//to Garlic
      O     "Blend_T-41".Dose_Garlic.QDOSERun;  //Dose Run
      =     "Blend to Preparation"."T-41".Raw_Material.Garlic.DoseRun;
      O     "Blend_T-41".Dose_Garlic.QHELD;  //Dose Held
      =     "Blend to Preparation"."T-41".Raw_Material.Garlic.DoseHeld;
      O     "Blend_T-41".Dose_Garlic.QDoseComplete;  //Dose Complete
      =     "Blend to Preparation"."T-41".Raw_Material.Garlic.DoseComplete;
      O     "Blend_T-41".Dose_Garlic.V_CMD;  //Valve Command
      =     "Blend to Preparation"."T-41".Raw_Material.Garlic.ValveCMD;
      O     "Blend_T-41".Dose_Garlic.P_CMD;  //Pump Command
      =     "Blend to Preparation"."T-41".Raw_Material.Garlic.PumpCMD;
      O     "Blend_T-41".Dose.Dose_Header_Req.%X7;  //Header 1 Req
      =     "Blend to Preparation"."T-41".Raw_Material.Garlic.Header1_Req;
      O     "Blend_T-41".Dose.Dose_Header_Req.%X23;  //Header 2 Req
      =     "Blend to Preparation"."T-41".Raw_Material.Garlic.Header2_Req;
      L     "Blend to Preparation".Recipe."T-41".Garlic.Sp_DoseQty;  //Load Sp Dose From Recipe
      T     "Blend_T-41".SP_Garlic.Dose_SP;
      L     "Blend_T-41".Dose_Garlic.P_SPEED;  //Pump Speed
      T     "Blend to Preparation".Recipe."T-41".Garlic.SP_PumpSpeed;

//to Vinegar
      O     "Blend_T-41".Dose_Vinegar.QDOSERun;  //Dose Run
      =     "Blend to Preparation"."T-41".Raw_Material.Vinegar.DoseRun;
      O     "Blend_T-41".Dose_Vinegar.QHELD;  //Dose Held
      =     "Blend to Preparation"."T-41".Raw_Material.Vinegar.DoseHeld;
      O     "Blend_T-41".Dose_Vinegar.QDoseComplete;  //Dose Complete
      =     "Blend to Preparation"."T-41".Raw_Material.Vinegar.DoseComplete;
      O     "Blend_T-41".Dose_Vinegar.V_CMD;  //Valve Command
      =     "Blend to Preparation"."T-41".Raw_Material.Vinegar.ValveCMD;
      O     "Blend_T-41".Dose_Vinegar.P_CMD;  //Pump Command
      =     "Blend to Preparation"."T-41".Raw_Material.Vinegar.PumpCMD;
      L     "Blend to Preparation".Recipe."T-41".Vinegar.Sp_DoseQty;  //Load Sp Dose From Recipe
      T     "Blend_T-41".SP_Vinegar.Dose_SP;
      L     "Blend_T-41".Dose_Vinegar.P_SPEED;  //Pump Speed
      T     "Blend to Preparation".Recipe."T-41".Vinegar.SP_PumpSpeed;

//to HW
      O     "Blend_T-41".Dose_HW.QDOSERun;  //Dose Run
      =     "Blend to Preparation"."T-41".Raw_Material.HW.DoseRun;
      O     "Blend_T-41".Dose_HW.QHELD;  //Dose Held
      =     "Blend to Preparation"."T-41".Raw_Material.HW.DoseHeld;
      O     "Blend_T-41".Dose_HW.QDoseComplete;  //Dose Complete
      =     "Blend to Preparation"."T-41".Raw_Material.HW.DoseComplete;
      O     "Blend_T-41".Dose_HW.V_CMD;  //Valve Command
      =     "Blend to Preparation"."T-41".Raw_Material.HW.ValveCMD;
      O     "Blend_T-41".Dose_HW.P_CMD;  //Pump Command
      =     "Blend to Preparation"."T-41".Raw_Material.HW.PumpCMD;
      O     "Blend_T-41".Dose.Dose_Header_Req.%X8;  //Header 1 Req
      =     "Blend to Preparation"."T-41".Raw_Material.HW.Header1_Req;
      O     "Blend_T-41".Dose.Dose_Header_Req.%X24;  //Header 2 Req
      =     "Blend to Preparation"."T-41".Raw_Material.HW.Header2_Req;

      L     "Blend to Preparation".Recipe."T-41".HW.Sp_Flush_to_BlendQty;  //Load Flush to Blend Sp Dose From Recipe
      T     "Blend_T-41"."HW Flushing".Qty."Flush to Blend Qty";
      L     "Blend to Preparation".Recipe."T-41".HW.Sp_Flush_to_DrainQty;  //Load Flush to Blend Sp Dose From Recipe
      T     "Blend_T-41"."HW Flushing".Qty."Flush to Drain Qty";  //Load Drain Time from recipe
      L     "Blend to Preparation".Recipe."T-41".HW.Sp_DrainTime;
      T     "Blend_T-41"."HW Flushing".TimeDrain_SP;

      L     "Blend_T-41".Dose_HW.P_SPEED;  //Pump Speed
      T     "Blend to Preparation".Recipe."T-41".HW.SP_PumpSpeed;


//General
      O     "Blend_T-41".IN_FBAV_Header1;
      =     "Blend to Preparation"."T-41".LineHeader1_OK;
      O     "Blend_T-41".IN_FBAV_Header2;
      =     "Blend to Preparation"."T-41".LineHeader2_OK;
      O     "Blend_T-41".IN_FBAV_Vinegar;
      =     "Blend to Preparation"."T-41".LineVinegar_OK;


REGION Network 124: Comm to Salt
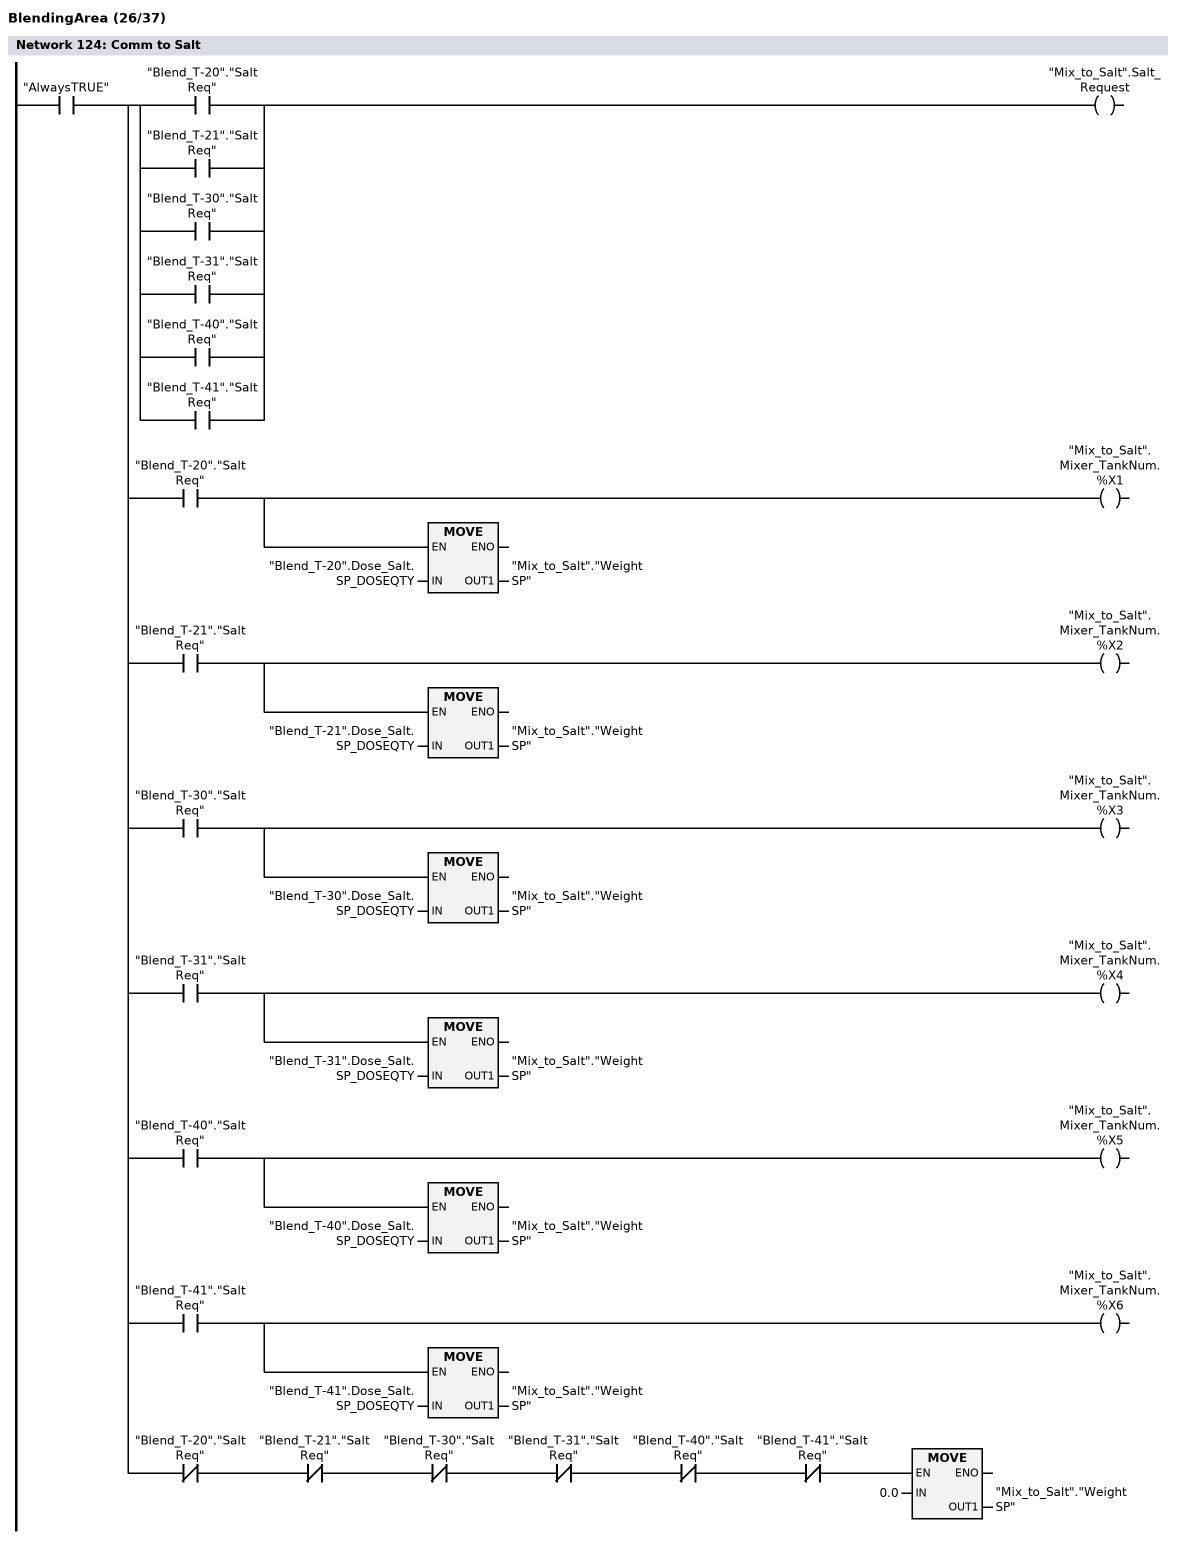
   RUNG wire#powerrail
      Contact( "AlwaysTRUE" )
      wire#w1
      Contact( "Blend_T-20"."Salt Req" )
      wire#w2
      Coil( "Mix_to_Salt".Salt_Request )
   END_RUNG
   RUNG wire#w1
      Contact( "Blend_T-21"."Salt Req" )
   END_RUNG wire#w2
   RUNG wire#w1
      Contact( "Blend_T-30"."Salt Req" )
   END_RUNG wire#w2
   RUNG wire#w1
      Contact( "Blend_T-31"."Salt Req" )
   END_RUNG wire#w2
   RUNG wire#w1
      Contact( "Blend_T-40"."Salt Req" )
   END_RUNG wire#w2
   RUNG wire#w1
      Contact( "Blend_T-41"."Salt Req" )
   END_RUNG wire#w2
   RUNG wire#w1
      Contact( "Blend_T-20"."Salt Req" )
      wire#w3
      Coil( "Mix_to_Salt".Mixer_TankNum.%X1 )
   END_RUNG
   RUNG wire#w3
      Move(in := "Blend_T-20".Dose_Salt.SP_DOSEQTY, out1 => "Mix_to_Salt"."Weight SP")
   END_RUNG
   RUNG wire#w1
      Contact( "Blend_T-21"."Salt Req" )
      wire#w4
      Coil( "Mix_to_Salt".Mixer_TankNum.%X2 )
   END_RUNG
   RUNG wire#w4
      Move(in := "Blend_T-21".Dose_Salt.SP_DOSEQTY, out1 => "Mix_to_Salt"."Weight SP")
   END_RUNG
   RUNG wire#w1
      Contact( "Blend_T-30"."Salt Req" )
      wire#w5
      Coil( "Mix_to_Salt".Mixer_TankNum.%X3 )
   END_RUNG
   RUNG wire#w5
      Move(in := "Blend_T-30".Dose_Salt.SP_DOSEQTY, out1 => "Mix_to_Salt"."Weight SP")
   END_RUNG
   RUNG wire#w1
      Contact( "Blend_T-31"."Salt Req" )
      wire#w6
      Coil( "Mix_to_Salt".Mixer_TankNum.%X4 )
   END_RUNG
   RUNG wire#w6
      Move(in := "Blend_T-31".Dose_Salt.SP_DOSEQTY, out1 => "Mix_to_Salt"."Weight SP")
   END_RUNG
   RUNG wire#w1
      Contact( "Blend_T-40"."Salt Req" )
      wire#w7
      Coil( "Mix_to_Salt".Mixer_TankNum.%X5 )
   END_RUNG
   RUNG wire#w7
      Move(in := "Blend_T-40".Dose_Salt.SP_DOSEQTY, out1 => "Mix_to_Salt"."Weight SP")
   END_RUNG
   RUNG wire#w1
      Contact( "Blend_T-41"."Salt Req" )
      wire#w8
      Coil( "Mix_to_Salt".Mixer_TankNum.%X6 )
   END_RUNG
   RUNG wire#w8
      Move(in := "Blend_T-41".Dose_Salt.SP_DOSEQTY, out1 => "Mix_to_Salt"."Weight SP")
   END_RUNG
   RUNG wire#w1
      I_Contact( "Blend_T-20"."Salt Req" )
      I_Contact( "Blend_T-21"."Salt Req" )
      I_Contact( "Blend_T-30"."Salt Req" )
      I_Contact( "Blend_T-31"."Salt Req" )
      I_Contact( "Blend_T-40"."Salt Req" )
      I_Contact( "Blend_T-41"."Salt Req" )
      Move(in := 0.0, out1 => "Mix_to_Salt"."Weight SP")
   END_RUNG
   // the same network as SCL:
   "Mix_to_Salt".Salt_Request := "AlwaysTRUE" AND ("Blend_T-20"."Salt Req" OR "Blend_T-21"."Salt Req" OR "Blend_T-30"."Salt Req" OR "Blend_T-31"."Salt Req" OR "Blend_T-40"."Salt Req" OR "Blend_T-41"."Salt Req");
   "Mix_to_Salt".Mixer_TankNum.%X1 := "AlwaysTRUE" AND "Blend_T-20"."Salt Req";
   IF "Mix_to_Salt".Mixer_TankNum.%X1 THEN
       "Mix_to_Salt"."Weight SP" := "Blend_T-20".Dose_Salt.SP_DOSEQTY;
   END_IF;
   "Mix_to_Salt".Mixer_TankNum.%X2 := "AlwaysTRUE" AND "Blend_T-21"."Salt Req";
   IF "Mix_to_Salt".Mixer_TankNum.%X2 THEN
       "Mix_to_Salt"."Weight SP" := "Blend_T-21".Dose_Salt.SP_DOSEQTY;
   END_IF;
   "Mix_to_Salt".Mixer_TankNum.%X3 := "AlwaysTRUE" AND "Blend_T-30"."Salt Req";
   IF "Mix_to_Salt".Mixer_TankNum.%X3 THEN
       "Mix_to_Salt"."Weight SP" := "Blend_T-30".Dose_Salt.SP_DOSEQTY;
   END_IF;
   "Mix_to_Salt".Mixer_TankNum.%X4 := "AlwaysTRUE" AND "Blend_T-31"."Salt Req";
   IF "Mix_to_Salt".Mixer_TankNum.%X4 THEN
       "Mix_to_Salt"."Weight SP" := "Blend_T-31".Dose_Salt.SP_DOSEQTY;
   END_IF;
   "Mix_to_Salt".Mixer_TankNum.%X5 := "AlwaysTRUE" AND "Blend_T-40"."Salt Req";
   IF "Mix_to_Salt".Mixer_TankNum.%X5 THEN
       "Mix_to_Salt"."Weight SP" := "Blend_T-40".Dose_Salt.SP_DOSEQTY;
   END_IF;
   "Mix_to_Salt".Mixer_TankNum.%X6 := "AlwaysTRUE" AND "Blend_T-41"."Salt Req";
   IF "Mix_to_Salt".Mixer_TankNum.%X6 THEN
       "Mix_to_Salt"."Weight SP" := "Blend_T-41".Dose_Salt.SP_DOSEQTY;
   END_IF;
   IF "AlwaysTRUE" AND NOT "Blend_T-20"."Salt Req" AND NOT "Blend_T-21"."Salt Req" AND NOT "Blend_T-30"."Salt Req" AND NOT "Blend_T-31"."Salt Req" AND NOT "Blend_T-40"."Salt Req" AND NOT "Blend_T-41"."Salt Req" THEN
       "Mix_to_Salt"."Weight SP" := 0.0;
   END_IF;
END_REGION

REGION Network 125: Comm to Sugar
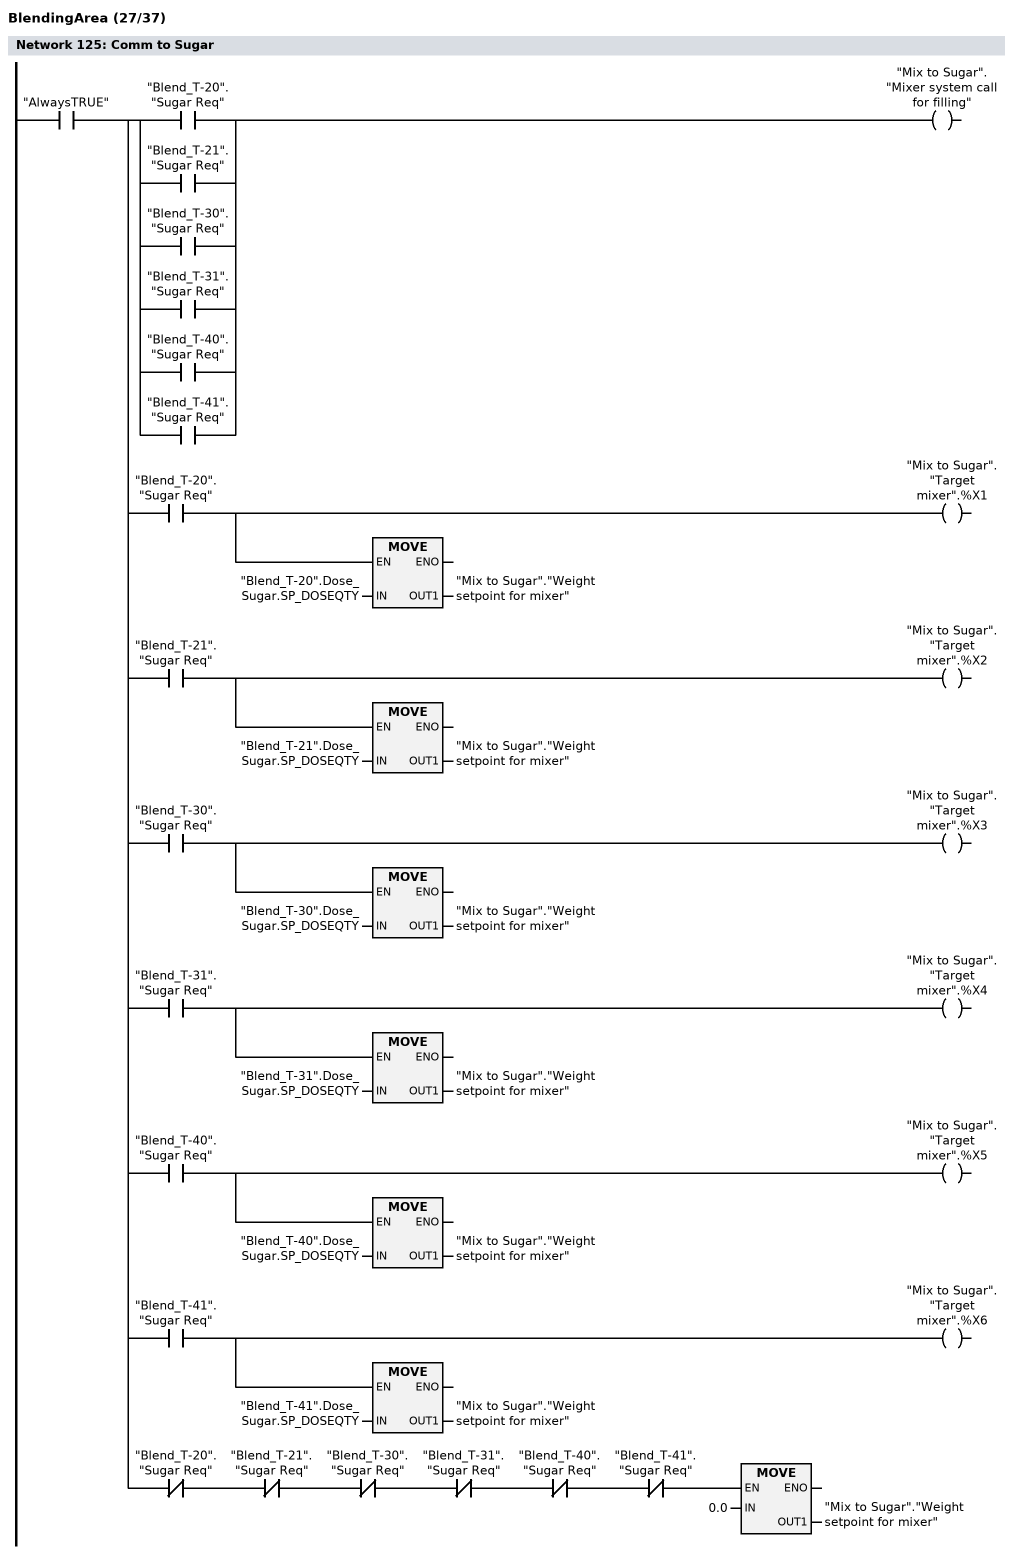
   RUNG wire#powerrail
      Contact( "AlwaysTRUE" )
      wire#w1
      Contact( "Blend_T-20"."Sugar Req" )
      wire#w2
      Coil( "Mix to Sugar"."Mixer system call for filling" )
   END_RUNG
   RUNG wire#w1
      Contact( "Blend_T-21"."Sugar Req" )
   END_RUNG wire#w2
   RUNG wire#w1
      Contact( "Blend_T-30"."Sugar Req" )
   END_RUNG wire#w2
   RUNG wire#w1
      Contact( "Blend_T-31"."Sugar Req" )
   END_RUNG wire#w2
   RUNG wire#w1
      Contact( "Blend_T-40"."Sugar Req" )
   END_RUNG wire#w2
   RUNG wire#w1
      Contact( "Blend_T-41"."Sugar Req" )
   END_RUNG wire#w2
   RUNG wire#w1
      Contact( "Blend_T-20"."Sugar Req" )
      wire#w3
      Coil( "Mix to Sugar"."Target mixer".%X1 )
   END_RUNG
   RUNG wire#w3
      Move(in := "Blend_T-20".Dose_Sugar.SP_DOSEQTY, out1 => "Mix to Sugar"."Weight setpoint for mixer")
   END_RUNG
   RUNG wire#w1
      Contact( "Blend_T-21"."Sugar Req" )
      wire#w4
      Coil( "Mix to Sugar"."Target mixer".%X2 )
   END_RUNG
   RUNG wire#w4
      Move(in := "Blend_T-21".Dose_Sugar.SP_DOSEQTY, out1 => "Mix to Sugar"."Weight setpoint for mixer")
   END_RUNG
   RUNG wire#w1
      Contact( "Blend_T-30"."Sugar Req" )
      wire#w5
      Coil( "Mix to Sugar"."Target mixer".%X3 )
   END_RUNG
   RUNG wire#w5
      Move(in := "Blend_T-30".Dose_Sugar.SP_DOSEQTY, out1 => "Mix to Sugar"."Weight setpoint for mixer")
   END_RUNG
   RUNG wire#w1
      Contact( "Blend_T-31"."Sugar Req" )
      wire#w6
      Coil( "Mix to Sugar"."Target mixer".%X4 )
   END_RUNG
   RUNG wire#w6
      Move(in := "Blend_T-31".Dose_Sugar.SP_DOSEQTY, out1 => "Mix to Sugar"."Weight setpoint for mixer")
   END_RUNG
   RUNG wire#w1
      Contact( "Blend_T-40"."Sugar Req" )
      wire#w7
      Coil( "Mix to Sugar"."Target mixer".%X5 )
   END_RUNG
   RUNG wire#w7
      Move(in := "Blend_T-40".Dose_Sugar.SP_DOSEQTY, out1 => "Mix to Sugar"."Weight setpoint for mixer")
   END_RUNG
   RUNG wire#w1
      Contact( "Blend_T-41"."Sugar Req" )
      wire#w8
      Coil( "Mix to Sugar"."Target mixer".%X6 )
   END_RUNG
   RUNG wire#w8
      Move(in := "Blend_T-41".Dose_Sugar.SP_DOSEQTY, out1 => "Mix to Sugar"."Weight setpoint for mixer")
   END_RUNG
   RUNG wire#w1
      I_Contact( "Blend_T-20"."Sugar Req" )
      I_Contact( "Blend_T-21"."Sugar Req" )
      I_Contact( "Blend_T-30"."Sugar Req" )
      I_Contact( "Blend_T-31"."Sugar Req" )
      I_Contact( "Blend_T-40"."Sugar Req" )
      I_Contact( "Blend_T-41"."Sugar Req" )
      Move(in := 0.0, out1 => "Mix to Sugar"."Weight setpoint for mixer")
   END_RUNG
   // the same network as SCL:
   "Mix to Sugar"."Mixer system call for filling" := "AlwaysTRUE" AND ("Blend_T-20"."Sugar Req" OR "Blend_T-21"."Sugar Req" OR "Blend_T-30"."Sugar Req" OR "Blend_T-31"."Sugar Req" OR "Blend_T-40"."Sugar Req" OR "Blend_T-41"."Sugar Req");
   "Mix to Sugar"."Target mixer".%X1 := "AlwaysTRUE" AND "Blend_T-20"."Sugar Req";
   IF "Mix to Sugar"."Target mixer".%X1 THEN
       "Mix to Sugar"."Weight setpoint for mixer" := "Blend_T-20".Dose_Sugar.SP_DOSEQTY;
   END_IF;
   "Mix to Sugar"."Target mixer".%X2 := "AlwaysTRUE" AND "Blend_T-21"."Sugar Req";
   IF "Mix to Sugar"."Target mixer".%X2 THEN
       "Mix to Sugar"."Weight setpoint for mixer" := "Blend_T-21".Dose_Sugar.SP_DOSEQTY;
   END_IF;
   "Mix to Sugar"."Target mixer".%X3 := "AlwaysTRUE" AND "Blend_T-30"."Sugar Req";
   IF "Mix to Sugar"."Target mixer".%X3 THEN
       "Mix to Sugar"."Weight setpoint for mixer" := "Blend_T-30".Dose_Sugar.SP_DOSEQTY;
   END_IF;
   "Mix to Sugar"."Target mixer".%X4 := "AlwaysTRUE" AND "Blend_T-31"."Sugar Req";
   IF "Mix to Sugar"."Target mixer".%X4 THEN
       "Mix to Sugar"."Weight setpoint for mixer" := "Blend_T-31".Dose_Sugar.SP_DOSEQTY;
   END_IF;
   "Mix to Sugar"."Target mixer".%X5 := "AlwaysTRUE" AND "Blend_T-40"."Sugar Req";
   IF "Mix to Sugar"."Target mixer".%X5 THEN
       "Mix to Sugar"."Weight setpoint for mixer" := "Blend_T-40".Dose_Sugar.SP_DOSEQTY;
   END_IF;
   "Mix to Sugar"."Target mixer".%X6 := "AlwaysTRUE" AND "Blend_T-41"."Sugar Req";
   IF "Mix to Sugar"."Target mixer".%X6 THEN
       "Mix to Sugar"."Weight setpoint for mixer" := "Blend_T-41".Dose_Sugar.SP_DOSEQTY;
   END_IF;
   IF "AlwaysTRUE" AND NOT "Blend_T-20"."Sugar Req" AND NOT "Blend_T-21"."Sugar Req" AND NOT "Blend_T-30"."Sugar Req" AND NOT "Blend_T-31"."Sugar Req" AND NOT "Blend_T-40"."Sugar Req" AND NOT "Blend_T-41"."Sugar Req" THEN
       "Mix to Sugar"."Weight setpoint for mixer" := 0.0;
   END_IF;
END_REGION

REGION Network 127: Comm to Buffer Tank THE 5
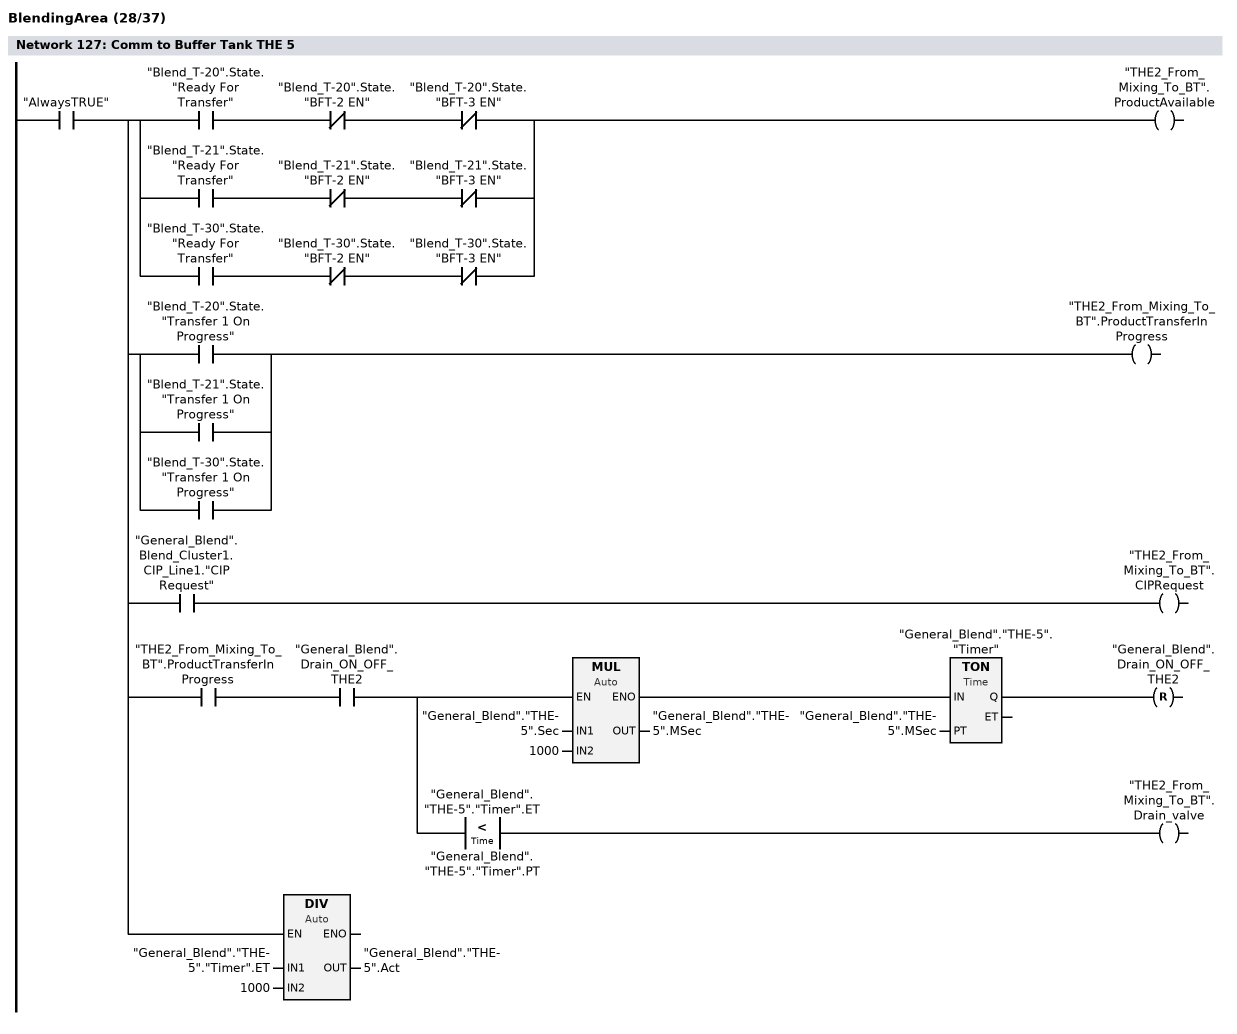
   RUNG wire#powerrail
      Contact( "AlwaysTRUE" )
      wire#w1
      Contact( "Blend_T-20".State."Ready For Transfer" )
      I_Contact( "Blend_T-20".State."BFT-2 EN" )
      I_Contact( "Blend_T-20".State."BFT-3 EN" )
      wire#w2
      Coil( "THE2_From_Mixing_To_BT".ProductAvailable )
   END_RUNG
   RUNG wire#w1
      Contact( "Blend_T-21".State."Ready For Transfer" )
      I_Contact( "Blend_T-21".State."BFT-2 EN" )
      I_Contact( "Blend_T-21".State."BFT-3 EN" )
   END_RUNG wire#w2
   RUNG wire#w1
      Contact( "Blend_T-30".State."Ready For Transfer" )
      I_Contact( "Blend_T-30".State."BFT-2 EN" )
      I_Contact( "Blend_T-30".State."BFT-3 EN" )
   END_RUNG wire#w2
   RUNG wire#w1
      Contact( "Blend_T-20".State."Transfer 1 On Progress" )
      wire#w3
      Coil( "THE2_From_Mixing_To_BT".ProductTransferInProgress )
   END_RUNG
   RUNG wire#w1
      Contact( "Blend_T-21".State."Transfer 1 On Progress" )
   END_RUNG wire#w3
   RUNG wire#w1
      Contact( "Blend_T-30".State."Transfer 1 On Progress" )
   END_RUNG wire#w3
   RUNG wire#w1
      Contact( "General_Blend".Blend_Cluster1.CIP_Line1."CIP Request" )
      Coil( "THE2_From_Mixing_To_BT".CIPRequest )
   END_RUNG
   RUNG wire#w1
      Contact( "THE2_From_Mixing_To_BT".ProductTransferInProgress )
      Contact( "General_Blend".Drain_ON_OFF_THE2 )
      wire#w4
      Mul(in1 := "General_Blend"."THE-5".Sec, in2 := 1000, out => "General_Blend"."THE-5".MSec)
      { S7_Templates := "time_type := Time" } "General_Blend"."THE-5"."Timer".TON(pt := "General_Blend"."THE-5".MSec, et =>)
      R_Coil( "General_Blend".Drain_ON_OFF_THE2 )
   END_RUNG
   RUNG wire#w4
      { S7_Templates := "SrcType := Time" } LT_Contact(in1 := "General_Blend"."THE-5"."Timer".ET, in2 := "General_Blend"."THE-5"."Timer".PT)
      Coil( "THE2_From_Mixing_To_BT".Drain_valve )
   END_RUNG
   RUNG wire#w1
      Div(in1 := "General_Blend"."THE-5"."Timer".ET, in2 := 1000, out => "General_Blend"."THE-5".Act)
   END_RUNG
   // the same network as SCL:
   "THE2_From_Mixing_To_BT".ProductAvailable := "AlwaysTRUE" AND (("Blend_T-20".State."Ready For Transfer" AND NOT "Blend_T-20".State."BFT-2 EN" AND NOT "Blend_T-20".State."BFT-3 EN") OR ("Blend_T-21".State."Ready For Transfer" AND NOT "Blend_T-21".State."BFT-2 EN" AND NOT "Blend_T-21".State."BFT-3 EN") OR ("Blend_T-30".State."Ready For Transfer" AND NOT "Blend_T-30".State."BFT-2 EN" AND NOT "Blend_T-30".State."BFT-3 EN"));
   "THE2_From_Mixing_To_BT".ProductTransferInProgress := "AlwaysTRUE" AND ("Blend_T-20".State."Transfer 1 On Progress" OR "Blend_T-21".State."Transfer 1 On Progress" OR "Blend_T-30".State."Transfer 1 On Progress");
   "THE2_From_Mixing_To_BT".CIPRequest := "AlwaysTRUE" AND "General_Blend".Blend_Cluster1.CIP_Line1."CIP Request";
   #_w1 := "AlwaysTRUE" AND "THE2_From_Mixing_To_BT".ProductTransferInProgress AND "General_Blend".Drain_ON_OFF_THE2;
   IF #_w1 THEN "General_Blend"."THE-5".MSec := "General_Blend"."THE-5".Sec * 1000; END_IF;
   "General_Blend"."THE-5"."Timer".TON(IN := #_w1, PT := "General_Blend"."THE-5".MSec);
   IF "General_Blend"."THE-5"."Timer".Q THEN "General_Blend".Drain_ON_OFF_THE2 := FALSE; END_IF;
   "THE2_From_Mixing_To_BT".Drain_valve := #_w1 AND ("General_Blend"."THE-5"."Timer".ET < "General_Blend"."THE-5"."Timer".PT);
   IF "AlwaysTRUE" THEN "General_Blend"."THE-5".Act := "General_Blend"."THE-5"."Timer".ET / 1000; END_IF;
END_REGION

REGION Network 128: Comm to Buffer Tank THE 4
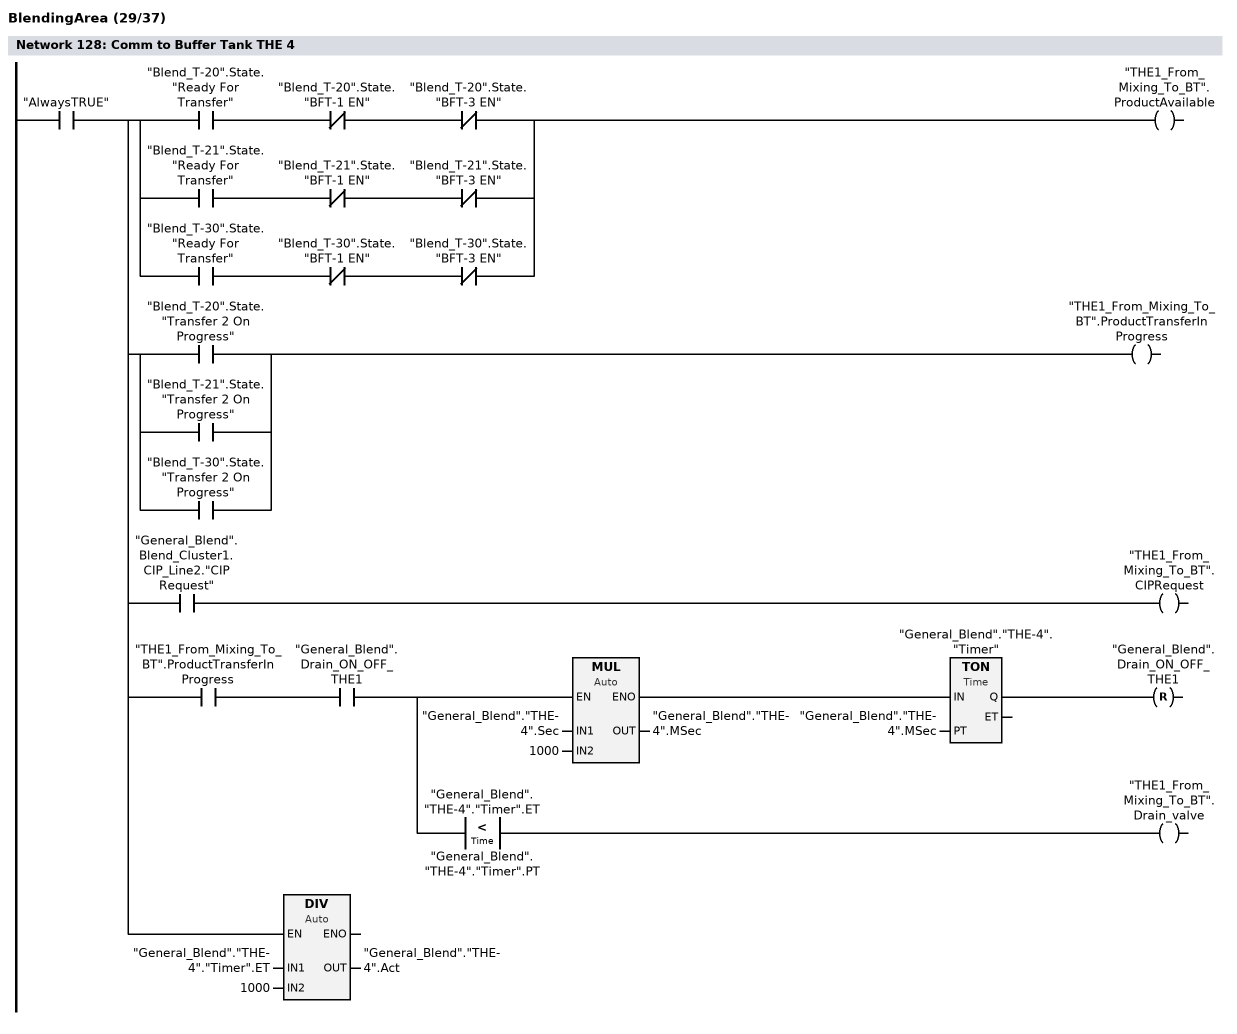
   RUNG wire#powerrail
      Contact( "AlwaysTRUE" )
      wire#w1
      Contact( "Blend_T-20".State."Ready For Transfer" )
      I_Contact( "Blend_T-20".State."BFT-1 EN" )
      I_Contact( "Blend_T-20".State."BFT-3 EN" )
      wire#w2
      Coil( "THE1_From_Mixing_To_BT".ProductAvailable )
   END_RUNG
   RUNG wire#w1
      Contact( "Blend_T-21".State."Ready For Transfer" )
      I_Contact( "Blend_T-21".State."BFT-1 EN" )
      I_Contact( "Blend_T-21".State."BFT-3 EN" )
   END_RUNG wire#w2
   RUNG wire#w1
      Contact( "Blend_T-30".State."Ready For Transfer" )
      I_Contact( "Blend_T-30".State."BFT-1 EN" )
      I_Contact( "Blend_T-30".State."BFT-3 EN" )
   END_RUNG wire#w2
   RUNG wire#w1
      Contact( "Blend_T-20".State."Transfer 2 On Progress" )
      wire#w3
      Coil( "THE1_From_Mixing_To_BT".ProductTransferInProgress )
   END_RUNG
   RUNG wire#w1
      Contact( "Blend_T-21".State."Transfer 2 On Progress" )
   END_RUNG wire#w3
   RUNG wire#w1
      Contact( "Blend_T-30".State."Transfer 2 On Progress" )
   END_RUNG wire#w3
   RUNG wire#w1
      Contact( "General_Blend".Blend_Cluster1.CIP_Line2."CIP Request" )
      Coil( "THE1_From_Mixing_To_BT".CIPRequest )
   END_RUNG
   RUNG wire#w1
      Contact( "THE1_From_Mixing_To_BT".ProductTransferInProgress )
      Contact( "General_Blend".Drain_ON_OFF_THE1 )
      wire#w4
      Mul(in1 := "General_Blend"."THE-4".Sec, in2 := 1000, out => "General_Blend"."THE-4".MSec)
      { S7_Templates := "time_type := Time" } "General_Blend"."THE-4"."Timer".TON(pt := "General_Blend"."THE-4".MSec, et =>)
      R_Coil( "General_Blend".Drain_ON_OFF_THE1 )
   END_RUNG
   RUNG wire#w4
      { S7_Templates := "SrcType := Time" } LT_Contact(in1 := "General_Blend"."THE-4"."Timer".ET, in2 := "General_Blend"."THE-4"."Timer".PT)
      Coil( "THE1_From_Mixing_To_BT".Drain_valve )
   END_RUNG
   RUNG wire#w1
      Div(in1 := "General_Blend"."THE-4"."Timer".ET, in2 := 1000, out => "General_Blend"."THE-4".Act)
   END_RUNG
   // the same network as SCL:
   "THE1_From_Mixing_To_BT".ProductAvailable := "AlwaysTRUE" AND (("Blend_T-20".State."Ready For Transfer" AND NOT "Blend_T-20".State."BFT-1 EN" AND NOT "Blend_T-20".State."BFT-3 EN") OR ("Blend_T-21".State."Ready For Transfer" AND NOT "Blend_T-21".State."BFT-1 EN" AND NOT "Blend_T-21".State."BFT-3 EN") OR ("Blend_T-30".State."Ready For Transfer" AND NOT "Blend_T-30".State."BFT-1 EN" AND NOT "Blend_T-30".State."BFT-3 EN"));
   "THE1_From_Mixing_To_BT".ProductTransferInProgress := "AlwaysTRUE" AND ("Blend_T-20".State."Transfer 2 On Progress" OR "Blend_T-21".State."Transfer 2 On Progress" OR "Blend_T-30".State."Transfer 2 On Progress");
   "THE1_From_Mixing_To_BT".CIPRequest := "AlwaysTRUE" AND "General_Blend".Blend_Cluster1.CIP_Line2."CIP Request";
   #_w1 := "AlwaysTRUE" AND "THE1_From_Mixing_To_BT".ProductTransferInProgress AND "General_Blend".Drain_ON_OFF_THE1;
   IF #_w1 THEN "General_Blend"."THE-4".MSec := "General_Blend"."THE-4".Sec * 1000; END_IF;
   "General_Blend"."THE-4"."Timer".TON(IN := #_w1, PT := "General_Blend"."THE-4".MSec);
   IF "General_Blend"."THE-4"."Timer".Q THEN "General_Blend".Drain_ON_OFF_THE1 := FALSE; END_IF;
   "THE1_From_Mixing_To_BT".Drain_valve := #_w1 AND ("General_Blend"."THE-4"."Timer".ET < "General_Blend"."THE-4"."Timer".PT);
   IF "AlwaysTRUE" THEN "General_Blend"."THE-4".Act := "General_Blend"."THE-4"."Timer".ET / 1000; END_IF;
END_REGION

REGION Network 130: Comm CIP to Blend 20
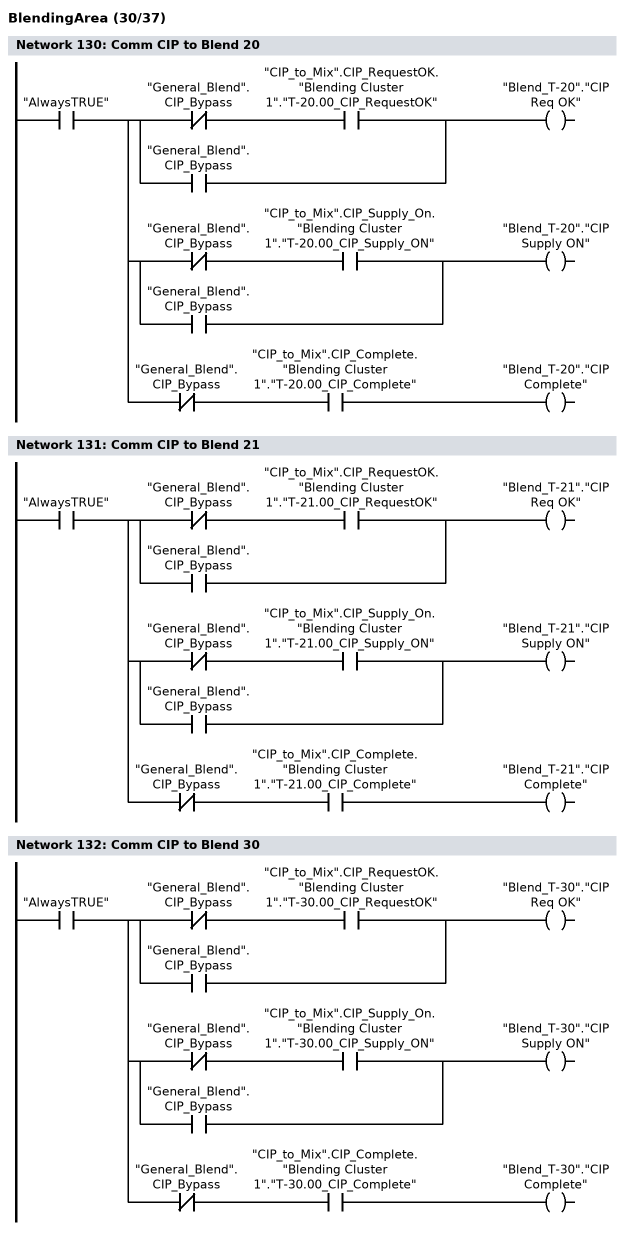
   RUNG wire#powerrail
      Contact( "AlwaysTRUE" )
      wire#w1
      I_Contact( "General_Blend".CIP_Bypass )
      Contact( "CIP_to_Mix".CIP_RequestOK."Blending Cluster 1"."T-20.00_CIP_RequestOK" )
      wire#w2
      Coil( "Blend_T-20"."CIP Req OK" )
   END_RUNG
   RUNG wire#w1
      Contact( "General_Blend".CIP_Bypass )
   END_RUNG wire#w2
   RUNG wire#w1
      I_Contact( "General_Blend".CIP_Bypass )
      Contact( "CIP_to_Mix".CIP_Supply_On."Blending Cluster 1"."T-20.00_CIP_Supply_ON" )
      wire#w3
      Coil( "Blend_T-20"."CIP Supply ON" )
   END_RUNG
   RUNG wire#w1
      Contact( "General_Blend".CIP_Bypass )
   END_RUNG wire#w3
   RUNG wire#w1
      I_Contact( "General_Blend".CIP_Bypass )
      Contact( "CIP_to_Mix".CIP_Complete."Blending Cluster 1"."T-20.00_CIP_Complete" )
      Coil( "Blend_T-20"."CIP Complete" )
   END_RUNG
   // the same network as SCL:
   "Blend_T-20"."CIP Req OK" := "AlwaysTRUE" AND ((NOT "General_Blend".CIP_Bypass AND "CIP_to_Mix".CIP_RequestOK."Blending Cluster 1"."T-20.00_CIP_RequestOK") OR "General_Blend".CIP_Bypass);
   "Blend_T-20"."CIP Supply ON" := "AlwaysTRUE" AND ((NOT "General_Blend".CIP_Bypass AND "CIP_to_Mix".CIP_Supply_On."Blending Cluster 1"."T-20.00_CIP_Supply_ON") OR "General_Blend".CIP_Bypass);
   "Blend_T-20"."CIP Complete" := "AlwaysTRUE" AND NOT "General_Blend".CIP_Bypass AND "CIP_to_Mix".CIP_Complete."Blending Cluster 1"."T-20.00_CIP_Complete";
END_REGION

REGION Network 131: Comm CIP to Blend 21
   RUNG wire#powerrail
      Contact( "AlwaysTRUE" )
      wire#w1
      I_Contact( "General_Blend".CIP_Bypass )
      Contact( "CIP_to_Mix".CIP_RequestOK."Blending Cluster 1"."T-21.00_CIP_RequestOK" )
      wire#w2
      Coil( "Blend_T-21"."CIP Req OK" )
   END_RUNG
   RUNG wire#w1
      Contact( "General_Blend".CIP_Bypass )
   END_RUNG wire#w2
   RUNG wire#w1
      I_Contact( "General_Blend".CIP_Bypass )
      Contact( "CIP_to_Mix".CIP_Supply_On."Blending Cluster 1"."T-21.00_CIP_Supply_ON" )
      wire#w3
      Coil( "Blend_T-21"."CIP Supply ON" )
   END_RUNG
   RUNG wire#w1
      Contact( "General_Blend".CIP_Bypass )
   END_RUNG wire#w3
   RUNG wire#w1
      I_Contact( "General_Blend".CIP_Bypass )
      Contact( "CIP_to_Mix".CIP_Complete."Blending Cluster 1"."T-21.00_CIP_Complete" )
      Coil( "Blend_T-21"."CIP Complete" )
   END_RUNG
   // the same network as SCL:
   "Blend_T-21"."CIP Req OK" := "AlwaysTRUE" AND ((NOT "General_Blend".CIP_Bypass AND "CIP_to_Mix".CIP_RequestOK."Blending Cluster 1"."T-21.00_CIP_RequestOK") OR "General_Blend".CIP_Bypass);
   "Blend_T-21"."CIP Supply ON" := "AlwaysTRUE" AND ((NOT "General_Blend".CIP_Bypass AND "CIP_to_Mix".CIP_Supply_On."Blending Cluster 1"."T-21.00_CIP_Supply_ON") OR "General_Blend".CIP_Bypass);
   "Blend_T-21"."CIP Complete" := "AlwaysTRUE" AND NOT "General_Blend".CIP_Bypass AND "CIP_to_Mix".CIP_Complete."Blending Cluster 1"."T-21.00_CIP_Complete";
END_REGION

REGION Network 132: Comm CIP to Blend 30
   RUNG wire#powerrail
      Contact( "AlwaysTRUE" )
      wire#w1
      I_Contact( "General_Blend".CIP_Bypass )
      Contact( "CIP_to_Mix".CIP_RequestOK."Blending Cluster 1"."T-30.00_CIP_RequestOK" )
      wire#w2
      Coil( "Blend_T-30"."CIP Req OK" )
   END_RUNG
   RUNG wire#w1
      Contact( "General_Blend".CIP_Bypass )
   END_RUNG wire#w2
   RUNG wire#w1
      I_Contact( "General_Blend".CIP_Bypass )
      Contact( "CIP_to_Mix".CIP_Supply_On."Blending Cluster 1"."T-30.00_CIP_Supply_ON" )
      wire#w3
      Coil( "Blend_T-30"."CIP Supply ON" )
   END_RUNG
   RUNG wire#w1
      Contact( "General_Blend".CIP_Bypass )
   END_RUNG wire#w3
   RUNG wire#w1
      I_Contact( "General_Blend".CIP_Bypass )
      Contact( "CIP_to_Mix".CIP_Complete."Blending Cluster 1"."T-30.00_CIP_Complete" )
      Coil( "Blend_T-30"."CIP Complete" )
   END_RUNG
   // the same network as SCL:
   "Blend_T-30"."CIP Req OK" := "AlwaysTRUE" AND ((NOT "General_Blend".CIP_Bypass AND "CIP_to_Mix".CIP_RequestOK."Blending Cluster 1"."T-30.00_CIP_RequestOK") OR "General_Blend".CIP_Bypass);
   "Blend_T-30"."CIP Supply ON" := "AlwaysTRUE" AND ((NOT "General_Blend".CIP_Bypass AND "CIP_to_Mix".CIP_Supply_On."Blending Cluster 1"."T-30.00_CIP_Supply_ON") OR "General_Blend".CIP_Bypass);
   "Blend_T-30"."CIP Complete" := "AlwaysTRUE" AND NOT "General_Blend".CIP_Bypass AND "CIP_to_Mix".CIP_Complete."Blending Cluster 1"."T-30.00_CIP_Complete";
END_REGION

REGION Network 133: Comm CIP to Blend 31
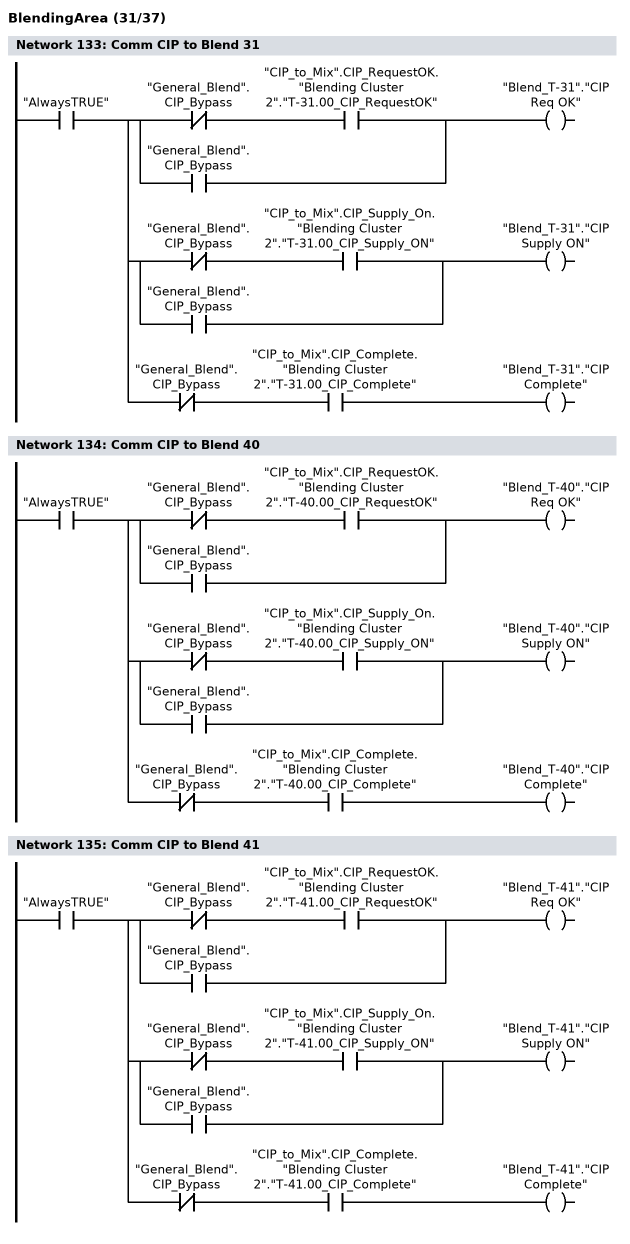
   RUNG wire#powerrail
      Contact( "AlwaysTRUE" )
      wire#w1
      I_Contact( "General_Blend".CIP_Bypass )
      Contact( "CIP_to_Mix".CIP_RequestOK."Blending Cluster 2"."T-31.00_CIP_RequestOK" )
      wire#w2
      Coil( "Blend_T-31"."CIP Req OK" )
   END_RUNG
   RUNG wire#w1
      Contact( "General_Blend".CIP_Bypass )
   END_RUNG wire#w2
   RUNG wire#w1
      I_Contact( "General_Blend".CIP_Bypass )
      Contact( "CIP_to_Mix".CIP_Supply_On."Blending Cluster 2"."T-31.00_CIP_Supply_ON" )
      wire#w3
      Coil( "Blend_T-31"."CIP Supply ON" )
   END_RUNG
   RUNG wire#w1
      Contact( "General_Blend".CIP_Bypass )
   END_RUNG wire#w3
   RUNG wire#w1
      I_Contact( "General_Blend".CIP_Bypass )
      Contact( "CIP_to_Mix".CIP_Complete."Blending Cluster 2"."T-31.00_CIP_Complete" )
      Coil( "Blend_T-31"."CIP Complete" )
   END_RUNG
   // the same network as SCL:
   "Blend_T-31"."CIP Req OK" := "AlwaysTRUE" AND ((NOT "General_Blend".CIP_Bypass AND "CIP_to_Mix".CIP_RequestOK."Blending Cluster 2"."T-31.00_CIP_RequestOK") OR "General_Blend".CIP_Bypass);
   "Blend_T-31"."CIP Supply ON" := "AlwaysTRUE" AND ((NOT "General_Blend".CIP_Bypass AND "CIP_to_Mix".CIP_Supply_On."Blending Cluster 2"."T-31.00_CIP_Supply_ON") OR "General_Blend".CIP_Bypass);
   "Blend_T-31"."CIP Complete" := "AlwaysTRUE" AND NOT "General_Blend".CIP_Bypass AND "CIP_to_Mix".CIP_Complete."Blending Cluster 2"."T-31.00_CIP_Complete";
END_REGION

REGION Network 134: Comm CIP to Blend 40
   RUNG wire#powerrail
      Contact( "AlwaysTRUE" )
      wire#w1
      I_Contact( "General_Blend".CIP_Bypass )
      Contact( "CIP_to_Mix".CIP_RequestOK."Blending Cluster 2"."T-40.00_CIP_RequestOK" )
      wire#w2
      Coil( "Blend_T-40"."CIP Req OK" )
   END_RUNG
   RUNG wire#w1
      Contact( "General_Blend".CIP_Bypass )
   END_RUNG wire#w2
   RUNG wire#w1
      I_Contact( "General_Blend".CIP_Bypass )
      Contact( "CIP_to_Mix".CIP_Supply_On."Blending Cluster 2"."T-40.00_CIP_Supply_ON" )
      wire#w3
      Coil( "Blend_T-40"."CIP Supply ON" )
   END_RUNG
   RUNG wire#w1
      Contact( "General_Blend".CIP_Bypass )
   END_RUNG wire#w3
   RUNG wire#w1
      I_Contact( "General_Blend".CIP_Bypass )
      Contact( "CIP_to_Mix".CIP_Complete."Blending Cluster 2"."T-40.00_CIP_Complete" )
      Coil( "Blend_T-40"."CIP Complete" )
   END_RUNG
   // the same network as SCL:
   "Blend_T-40"."CIP Req OK" := "AlwaysTRUE" AND ((NOT "General_Blend".CIP_Bypass AND "CIP_to_Mix".CIP_RequestOK."Blending Cluster 2"."T-40.00_CIP_RequestOK") OR "General_Blend".CIP_Bypass);
   "Blend_T-40"."CIP Supply ON" := "AlwaysTRUE" AND ((NOT "General_Blend".CIP_Bypass AND "CIP_to_Mix".CIP_Supply_On."Blending Cluster 2"."T-40.00_CIP_Supply_ON") OR "General_Blend".CIP_Bypass);
   "Blend_T-40"."CIP Complete" := "AlwaysTRUE" AND NOT "General_Blend".CIP_Bypass AND "CIP_to_Mix".CIP_Complete."Blending Cluster 2"."T-40.00_CIP_Complete";
END_REGION

REGION Network 135: Comm CIP to Blend 41
   RUNG wire#powerrail
      Contact( "AlwaysTRUE" )
      wire#w1
      I_Contact( "General_Blend".CIP_Bypass )
      Contact( "CIP_to_Mix".CIP_RequestOK."Blending Cluster 2"."T-41.00_CIP_RequestOK" )
      wire#w2
      Coil( "Blend_T-41"."CIP Req OK" )
   END_RUNG
   RUNG wire#w1
      Contact( "General_Blend".CIP_Bypass )
   END_RUNG wire#w2
   RUNG wire#w1
      I_Contact( "General_Blend".CIP_Bypass )
      Contact( "CIP_to_Mix".CIP_Supply_On."Blending Cluster 2"."T-41.00_CIP_Supply_ON" )
      wire#w3
      Coil( "Blend_T-41"."CIP Supply ON" )
   END_RUNG
   RUNG wire#w1
      Contact( "General_Blend".CIP_Bypass )
   END_RUNG wire#w3
   RUNG wire#w1
      I_Contact( "General_Blend".CIP_Bypass )
      Contact( "CIP_to_Mix".CIP_Complete."Blending Cluster 2"."T-41.00_CIP_Complete" )
      Coil( "Blend_T-41"."CIP Complete" )
   END_RUNG
   // the same network as SCL:
   "Blend_T-41"."CIP Req OK" := "AlwaysTRUE" AND ((NOT "General_Blend".CIP_Bypass AND "CIP_to_Mix".CIP_RequestOK."Blending Cluster 2"."T-41.00_CIP_RequestOK") OR "General_Blend".CIP_Bypass);
   "Blend_T-41"."CIP Supply ON" := "AlwaysTRUE" AND ((NOT "General_Blend".CIP_Bypass AND "CIP_to_Mix".CIP_Supply_On."Blending Cluster 2"."T-41.00_CIP_Supply_ON") OR "General_Blend".CIP_Bypass);
   "Blend_T-41"."CIP Complete" := "AlwaysTRUE" AND NOT "General_Blend".CIP_Bypass AND "CIP_to_Mix".CIP_Complete."Blending Cluster 2"."T-41.00_CIP_Complete";
END_REGION

REGION Network 137: CIP Line Blending Cluster 1 Enable
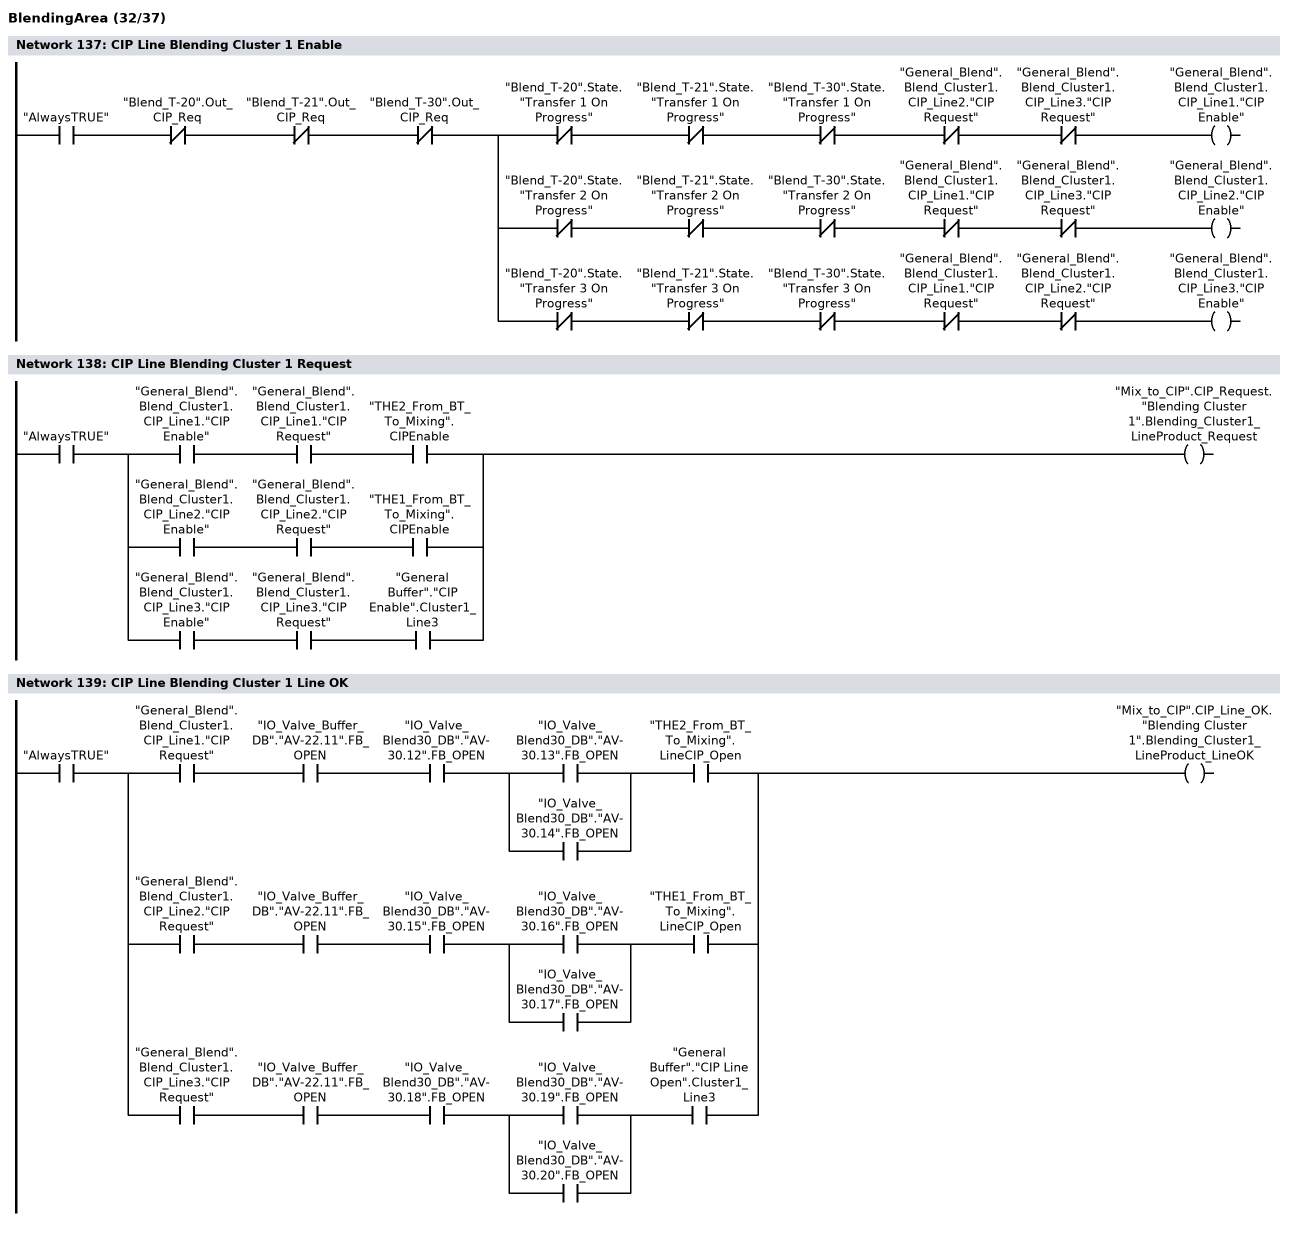
   RUNG wire#powerrail
      Contact( "AlwaysTRUE" )
      I_Contact( "Blend_T-20".Out_CIP_Req )
      I_Contact( "Blend_T-21".Out_CIP_Req )
      I_Contact( "Blend_T-30".Out_CIP_Req )
      wire#w1
      I_Contact( "Blend_T-20".State."Transfer 1 On Progress" )
      I_Contact( "Blend_T-21".State."Transfer 1 On Progress" )
      I_Contact( "Blend_T-30".State."Transfer 1 On Progress" )
      I_Contact( "General_Blend".Blend_Cluster1.CIP_Line2."CIP Request" )
      I_Contact( "General_Blend".Blend_Cluster1.CIP_Line3."CIP Request" )
      Coil( "General_Blend".Blend_Cluster1.CIP_Line1."CIP Enable" )
   END_RUNG
   RUNG wire#w1
      I_Contact( "Blend_T-20".State."Transfer 2 On Progress" )
      I_Contact( "Blend_T-21".State."Transfer 2 On Progress" )
      I_Contact( "Blend_T-30".State."Transfer 2 On Progress" )
      I_Contact( "General_Blend".Blend_Cluster1.CIP_Line1."CIP Request" )
      I_Contact( "General_Blend".Blend_Cluster1.CIP_Line3."CIP Request" )
      Coil( "General_Blend".Blend_Cluster1.CIP_Line2."CIP Enable" )
   END_RUNG
   RUNG wire#w1
      I_Contact( "Blend_T-20".State."Transfer 3 On Progress" )
      I_Contact( "Blend_T-21".State."Transfer 3 On Progress" )
      I_Contact( "Blend_T-30".State."Transfer 3 On Progress" )
      I_Contact( "General_Blend".Blend_Cluster1.CIP_Line1."CIP Request" )
      I_Contact( "General_Blend".Blend_Cluster1.CIP_Line2."CIP Request" )
      Coil( "General_Blend".Blend_Cluster1.CIP_Line3."CIP Enable" )
   END_RUNG
   // the same network as SCL:
   #_w1 := "AlwaysTRUE" AND NOT "Blend_T-20".Out_CIP_Req AND NOT "Blend_T-21".Out_CIP_Req AND NOT "Blend_T-30".Out_CIP_Req;
   "General_Blend".Blend_Cluster1.CIP_Line1."CIP Enable" := #_w1 AND NOT "Blend_T-20".State."Transfer 1 On Progress" AND NOT "Blend_T-21".State."Transfer 1 On Progress" AND NOT "Blend_T-30".State."Transfer 1 On Progress" AND NOT "General_Blend".Blend_Cluster1.CIP_Line2."CIP Request" AND NOT "General_Blend".Blend_Cluster1.CIP_Line3."CIP Request";
   "General_Blend".Blend_Cluster1.CIP_Line2."CIP Enable" := #_w1 AND NOT "Blend_T-20".State."Transfer 2 On Progress" AND NOT "Blend_T-21".State."Transfer 2 On Progress" AND NOT "Blend_T-30".State."Transfer 2 On Progress" AND NOT "General_Blend".Blend_Cluster1.CIP_Line1."CIP Request" AND NOT "General_Blend".Blend_Cluster1.CIP_Line3."CIP Request";
   "General_Blend".Blend_Cluster1.CIP_Line3."CIP Enable" := #_w1 AND NOT "Blend_T-20".State."Transfer 3 On Progress" AND NOT "Blend_T-21".State."Transfer 3 On Progress" AND NOT "Blend_T-30".State."Transfer 3 On Progress" AND NOT "General_Blend".Blend_Cluster1.CIP_Line1."CIP Request" AND NOT "General_Blend".Blend_Cluster1.CIP_Line2."CIP Request";
END_REGION

REGION Network 138: CIP Line Blending Cluster 1 Request
   RUNG wire#powerrail
      Contact( "AlwaysTRUE" )
      wire#w1
      Contact( "General_Blend".Blend_Cluster1.CIP_Line1."CIP Enable" )
      Contact( "General_Blend".Blend_Cluster1.CIP_Line1."CIP Request" )
      Contact( "THE2_From_BT_To_Mixing".CIPEnable )
      wire#w2
      Coil( "Mix_to_CIP".CIP_Request."Blending Cluster 1".Blending_Cluster1_LineProduct_Request )
   END_RUNG
   RUNG wire#w1
      Contact( "General_Blend".Blend_Cluster1.CIP_Line2."CIP Enable" )
      Contact( "General_Blend".Blend_Cluster1.CIP_Line2."CIP Request" )
      Contact( "THE1_From_BT_To_Mixing".CIPEnable )
   END_RUNG wire#w2
   RUNG wire#w1
      Contact( "General_Blend".Blend_Cluster1.CIP_Line3."CIP Enable" )
      Contact( "General_Blend".Blend_Cluster1.CIP_Line3."CIP Request" )
      Contact( "General Buffer"."CIP Enable".Cluster1_Line3 )
   END_RUNG wire#w2
   // the same network as SCL:
   "Mix_to_CIP".CIP_Request."Blending Cluster 1".Blending_Cluster1_LineProduct_Request := "AlwaysTRUE" AND (("General_Blend".Blend_Cluster1.CIP_Line1."CIP Enable" AND "General_Blend".Blend_Cluster1.CIP_Line1."CIP Request" AND "THE2_From_BT_To_Mixing".CIPEnable) OR ("General_Blend".Blend_Cluster1.CIP_Line2."CIP Enable" AND "General_Blend".Blend_Cluster1.CIP_Line2."CIP Request" AND "THE1_From_BT_To_Mixing".CIPEnable) OR ("General_Blend".Blend_Cluster1.CIP_Line3."CIP Enable" AND "General_Blend".Blend_Cluster1.CIP_Line3."CIP Request" AND "General Buffer"."CIP Enable".Cluster1_Line3));
END_REGION

REGION Network 139: CIP Line Blending Cluster 1 Line OK
   RUNG wire#powerrail
      Contact( "AlwaysTRUE" )
      wire#w1
      Contact( "General_Blend".Blend_Cluster1.CIP_Line1."CIP Request" )
      Contact( "IO_Valve_Buffer_DB"."AV-22.11".FB_OPEN )
      Contact( "IO_Valve_Blend30_DB"."AV-30.12".FB_OPEN )
      wire#w2
      Contact( "IO_Valve_Blend30_DB"."AV-30.13".FB_OPEN )
      wire#w3
      Contact( "THE2_From_BT_To_Mixing".LineCIP_Open )
      wire#w4
      Coil( "Mix_to_CIP".CIP_Line_OK."Blending Cluster 1".Blending_Cluster1_LineProduct_LineOK )
   END_RUNG
   RUNG wire#w2
      Contact( "IO_Valve_Blend30_DB"."AV-30.14".FB_OPEN )
   END_RUNG wire#w3
   RUNG wire#w1
      Contact( "General_Blend".Blend_Cluster1.CIP_Line2."CIP Request" )
      Contact( "IO_Valve_Buffer_DB"."AV-22.11".FB_OPEN )
      Contact( "IO_Valve_Blend30_DB"."AV-30.15".FB_OPEN )
      wire#w5
      Contact( "IO_Valve_Blend30_DB"."AV-30.16".FB_OPEN )
      wire#w6
      Contact( "THE1_From_BT_To_Mixing".LineCIP_Open )
   END_RUNG wire#w4
   RUNG wire#w5
      Contact( "IO_Valve_Blend30_DB"."AV-30.17".FB_OPEN )
   END_RUNG wire#w6
   RUNG wire#w1
      Contact( "General_Blend".Blend_Cluster1.CIP_Line3."CIP Request" )
      Contact( "IO_Valve_Buffer_DB"."AV-22.11".FB_OPEN )
      Contact( "IO_Valve_Blend30_DB"."AV-30.18".FB_OPEN )
      wire#w7
      Contact( "IO_Valve_Blend30_DB"."AV-30.19".FB_OPEN )
      wire#w8
      Contact( "General Buffer"."CIP Line Open".Cluster1_Line3 )
   END_RUNG wire#w4
   RUNG wire#w7
      Contact( "IO_Valve_Blend30_DB"."AV-30.20".FB_OPEN )
   END_RUNG wire#w8
   // the same network as SCL:
   "Mix_to_CIP".CIP_Line_OK."Blending Cluster 1".Blending_Cluster1_LineProduct_LineOK := "AlwaysTRUE" AND (("General_Blend".Blend_Cluster1.CIP_Line1."CIP Request" AND "IO_Valve_Buffer_DB"."AV-22.11".FB_OPEN AND "IO_Valve_Blend30_DB"."AV-30.12".FB_OPEN AND ("IO_Valve_Blend30_DB"."AV-30.13".FB_OPEN OR "IO_Valve_Blend30_DB"."AV-30.14".FB_OPEN) AND "THE2_From_BT_To_Mixing".LineCIP_Open) OR ("General_Blend".Blend_Cluster1.CIP_Line2."CIP Request" AND "IO_Valve_Buffer_DB"."AV-22.11".FB_OPEN AND "IO_Valve_Blend30_DB"."AV-30.15".FB_OPEN AND ("IO_Valve_Blend30_DB"."AV-30.16".FB_OPEN OR "IO_Valve_Blend30_DB"."AV-30.17".FB_OPEN) AND "THE1_From_BT_To_Mixing".LineCIP_Open) OR ("General_Blend".Blend_Cluster1.CIP_Line3."CIP Request" AND "IO_Valve_Buffer_DB"."AV-22.11".FB_OPEN AND "IO_Valve_Blend30_DB"."AV-30.18".FB_OPEN AND ("IO_Valve_Blend30_DB"."AV-30.19".FB_OPEN OR "IO_Valve_Blend30_DB"."AV-30.20".FB_OPEN) AND "General Buffer"."CIP Line Open".Cluster1_Line3));
END_REGION

REGION Network 140: CIP Line Blending Cluster 1 Valve Cmd
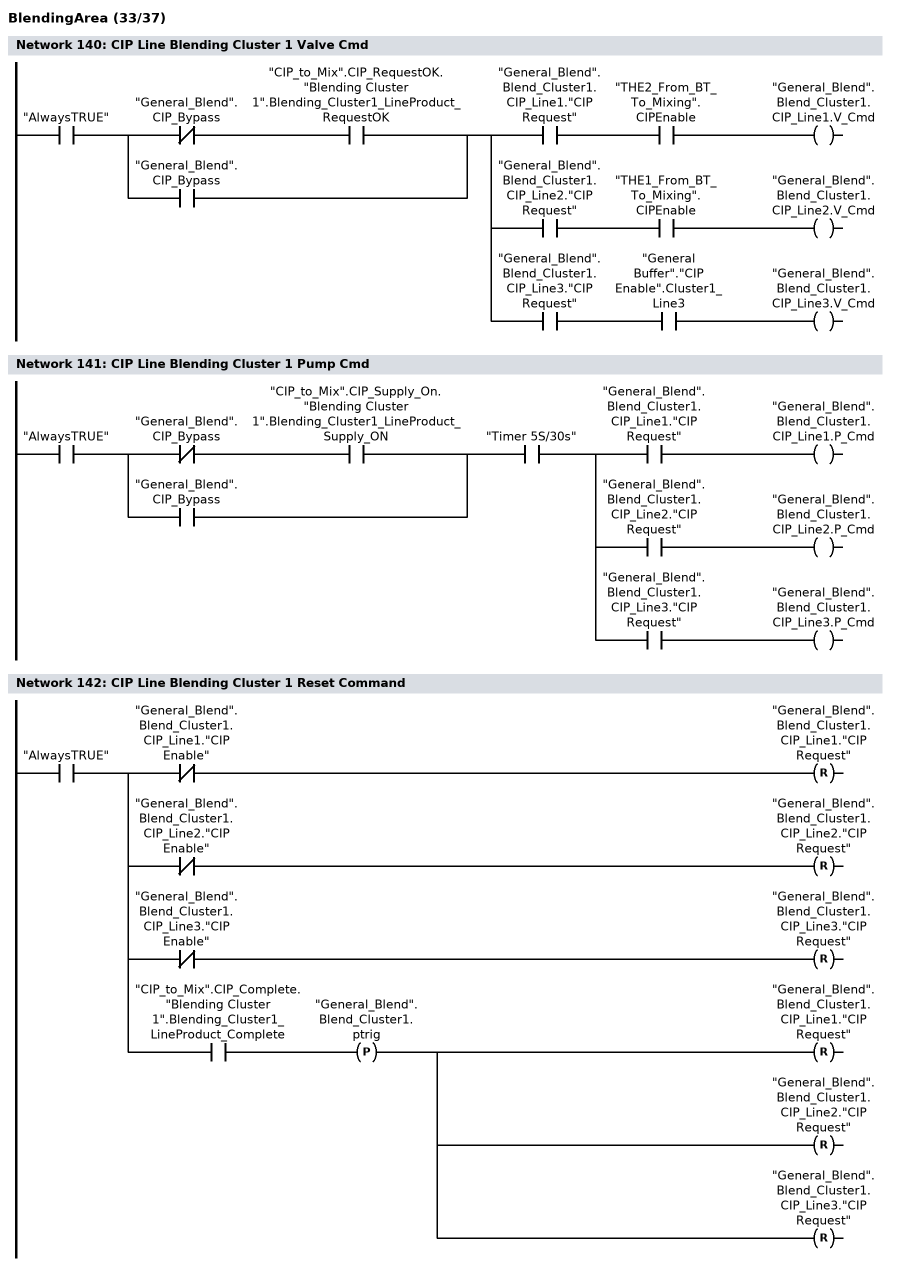
   RUNG wire#powerrail
      Contact( "AlwaysTRUE" )
      wire#w1
      I_Contact( "General_Blend".CIP_Bypass )
      Contact( "CIP_to_Mix".CIP_RequestOK."Blending Cluster 1".Blending_Cluster1_LineProduct_RequestOK )
      wire#w2
      Contact( "General_Blend".Blend_Cluster1.CIP_Line1."CIP Request" )
      Contact( "THE2_From_BT_To_Mixing".CIPEnable )
      Coil( "General_Blend".Blend_Cluster1.CIP_Line1.V_Cmd )
   END_RUNG
   RUNG wire#w1
      Contact( "General_Blend".CIP_Bypass )
   END_RUNG wire#w2
   RUNG wire#w2
      Contact( "General_Blend".Blend_Cluster1.CIP_Line2."CIP Request" )
      Contact( "THE1_From_BT_To_Mixing".CIPEnable )
      Coil( "General_Blend".Blend_Cluster1.CIP_Line2.V_Cmd )
   END_RUNG
   RUNG wire#w2
      Contact( "General_Blend".Blend_Cluster1.CIP_Line3."CIP Request" )
      Contact( "General Buffer"."CIP Enable".Cluster1_Line3 )
      Coil( "General_Blend".Blend_Cluster1.CIP_Line3.V_Cmd )
   END_RUNG
   // the same network as SCL:
   #_w1 := "AlwaysTRUE" AND ((NOT "General_Blend".CIP_Bypass AND "CIP_to_Mix".CIP_RequestOK."Blending Cluster 1".Blending_Cluster1_LineProduct_RequestOK) OR "General_Blend".CIP_Bypass);
   "General_Blend".Blend_Cluster1.CIP_Line1.V_Cmd := #_w1 AND "General_Blend".Blend_Cluster1.CIP_Line1."CIP Request" AND "THE2_From_BT_To_Mixing".CIPEnable;
   "General_Blend".Blend_Cluster1.CIP_Line2.V_Cmd := #_w1 AND "General_Blend".Blend_Cluster1.CIP_Line2."CIP Request" AND "THE1_From_BT_To_Mixing".CIPEnable;
   "General_Blend".Blend_Cluster1.CIP_Line3.V_Cmd := #_w1 AND "General_Blend".Blend_Cluster1.CIP_Line3."CIP Request" AND "General Buffer"."CIP Enable".Cluster1_Line3;
END_REGION

REGION Network 141: CIP Line Blending Cluster 1 Pump Cmd
   RUNG wire#powerrail
      Contact( "AlwaysTRUE" )
      wire#w1
      I_Contact( "General_Blend".CIP_Bypass )
      Contact( "CIP_to_Mix".CIP_Supply_On."Blending Cluster 1".Blending_Cluster1_LineProduct_Supply_ON )
      wire#w2
      Contact( "Timer 5S/30s" )
      wire#w3
      Contact( "General_Blend".Blend_Cluster1.CIP_Line1."CIP Request" )
      Coil( "General_Blend".Blend_Cluster1.CIP_Line1.P_Cmd )
   END_RUNG
   RUNG wire#w1
      Contact( "General_Blend".CIP_Bypass )
   END_RUNG wire#w2
   RUNG wire#w3
      Contact( "General_Blend".Blend_Cluster1.CIP_Line2."CIP Request" )
      Coil( "General_Blend".Blend_Cluster1.CIP_Line2.P_Cmd )
   END_RUNG
   RUNG wire#w3
      Contact( "General_Blend".Blend_Cluster1.CIP_Line3."CIP Request" )
      Coil( "General_Blend".Blend_Cluster1.CIP_Line3.P_Cmd )
   END_RUNG
   // the same network as SCL:
   #_w1 := "AlwaysTRUE" AND ((NOT "General_Blend".CIP_Bypass AND "CIP_to_Mix".CIP_Supply_On."Blending Cluster 1".Blending_Cluster1_LineProduct_Supply_ON) OR "General_Blend".CIP_Bypass) AND "Timer 5S/30s";
   "General_Blend".Blend_Cluster1.CIP_Line1.P_Cmd := #_w1 AND "General_Blend".Blend_Cluster1.CIP_Line1."CIP Request";
   "General_Blend".Blend_Cluster1.CIP_Line2.P_Cmd := #_w1 AND "General_Blend".Blend_Cluster1.CIP_Line2."CIP Request";
   "General_Blend".Blend_Cluster1.CIP_Line3.P_Cmd := #_w1 AND "General_Blend".Blend_Cluster1.CIP_Line3."CIP Request";
END_REGION

REGION Network 142: CIP Line Blending Cluster 1 Reset Command
   RUNG wire#powerrail
      Contact( "AlwaysTRUE" )
      wire#w1
      I_Contact( "General_Blend".Blend_Cluster1.CIP_Line1."CIP Enable" )
      R_Coil( "General_Blend".Blend_Cluster1.CIP_Line1."CIP Request" )
   END_RUNG
   RUNG wire#w1
      I_Contact( "General_Blend".Blend_Cluster1.CIP_Line2."CIP Enable" )
      R_Coil( "General_Blend".Blend_Cluster1.CIP_Line2."CIP Request" )
   END_RUNG
   RUNG wire#w1
      I_Contact( "General_Blend".Blend_Cluster1.CIP_Line3."CIP Enable" )
      R_Coil( "General_Blend".Blend_Cluster1.CIP_Line3."CIP Request" )
   END_RUNG
   RUNG wire#w1
      Contact( "CIP_to_Mix".CIP_Complete."Blending Cluster 1".Blending_Cluster1_LineProduct_Complete )
      P_Trig( "General_Blend".Blend_Cluster1.ptrig )
      wire#w2
      R_Coil( "General_Blend".Blend_Cluster1.CIP_Line1."CIP Request" )
   END_RUNG
   RUNG wire#w2
      R_Coil( "General_Blend".Blend_Cluster1.CIP_Line2."CIP Request" )
   END_RUNG
   RUNG wire#w2
      R_Coil( "General_Blend".Blend_Cluster1.CIP_Line3."CIP Request" )
   END_RUNG
   // the same network as SCL:
   IF "AlwaysTRUE" AND NOT "General_Blend".Blend_Cluster1.CIP_Line1."CIP Enable" THEN
       "General_Blend".Blend_Cluster1.CIP_Line1."CIP Request" := FALSE;
   END_IF;
   IF "AlwaysTRUE" AND NOT "General_Blend".Blend_Cluster1.CIP_Line2."CIP Enable" THEN
       "General_Blend".Blend_Cluster1.CIP_Line2."CIP Request" := FALSE;
   END_IF;
   IF "AlwaysTRUE" AND NOT "General_Blend".Blend_Cluster1.CIP_Line3."CIP Enable" THEN
       "General_Blend".Blend_Cluster1.CIP_Line3."CIP Request" := FALSE;
   END_IF;
   #_w1 := "AlwaysTRUE" AND "CIP_to_Mix".CIP_Complete."Blending Cluster 1".Blending_Cluster1_LineProduct_Complete;
   #_w2 := #_w1 AND NOT "General_Blend".Blend_Cluster1.ptrig;   // rising edge
   "General_Blend".Blend_Cluster1.ptrig := #_w1;
   IF #_w2 THEN
       "General_Blend".Blend_Cluster1.CIP_Line1."CIP Request" := FALSE;
       "General_Blend".Blend_Cluster1.CIP_Line2."CIP Request" := FALSE;
       "General_Blend".Blend_Cluster1.CIP_Line3."CIP Request" := FALSE;
   END_IF;
END_REGION

REGION Network 144: CIP Line Blending Cluster 2 Enable
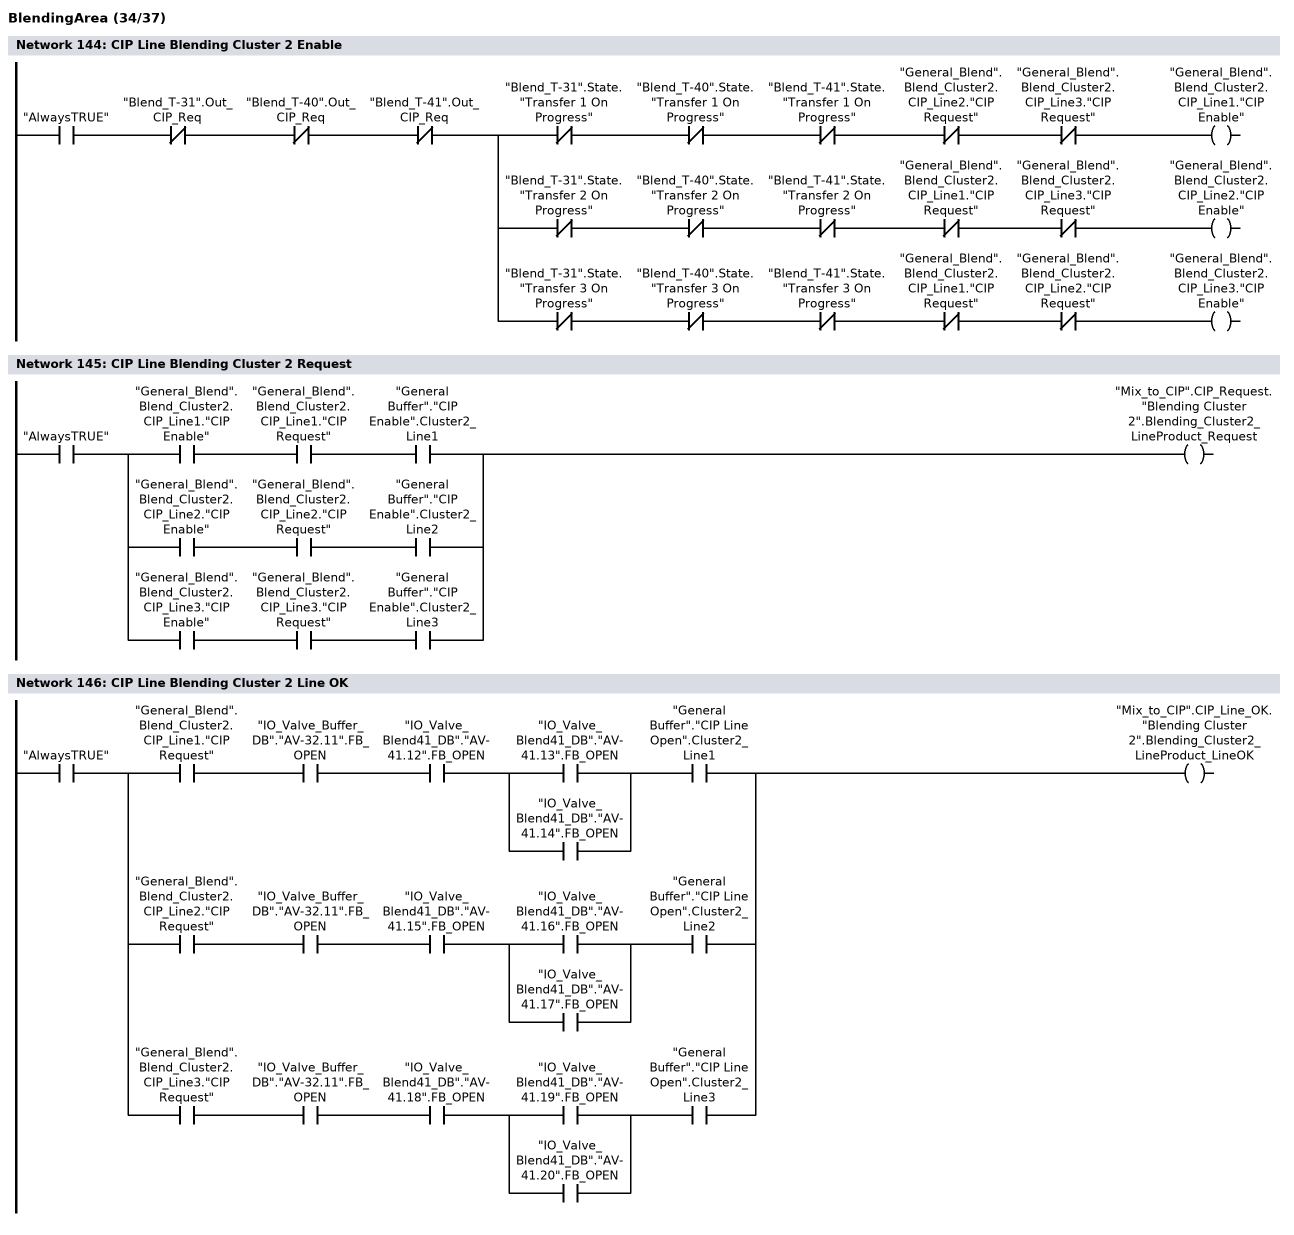
   RUNG wire#powerrail
      Contact( "AlwaysTRUE" )
      I_Contact( "Blend_T-31".Out_CIP_Req )
      I_Contact( "Blend_T-40".Out_CIP_Req )
      I_Contact( "Blend_T-41".Out_CIP_Req )
      wire#w1
      I_Contact( "Blend_T-31".State."Transfer 1 On Progress" )
      I_Contact( "Blend_T-40".State."Transfer 1 On Progress" )
      I_Contact( "Blend_T-41".State."Transfer 1 On Progress" )
      I_Contact( "General_Blend".Blend_Cluster2.CIP_Line2."CIP Request" )
      I_Contact( "General_Blend".Blend_Cluster2.CIP_Line3."CIP Request" )
      Coil( "General_Blend".Blend_Cluster2.CIP_Line1."CIP Enable" )
   END_RUNG
   RUNG wire#w1
      I_Contact( "Blend_T-31".State."Transfer 2 On Progress" )
      I_Contact( "Blend_T-40".State."Transfer 2 On Progress" )
      I_Contact( "Blend_T-41".State."Transfer 2 On Progress" )
      I_Contact( "General_Blend".Blend_Cluster2.CIP_Line1."CIP Request" )
      I_Contact( "General_Blend".Blend_Cluster2.CIP_Line3."CIP Request" )
      Coil( "General_Blend".Blend_Cluster2.CIP_Line2."CIP Enable" )
   END_RUNG
   RUNG wire#w1
      I_Contact( "Blend_T-31".State."Transfer 3 On Progress" )
      I_Contact( "Blend_T-40".State."Transfer 3 On Progress" )
      I_Contact( "Blend_T-41".State."Transfer 3 On Progress" )
      I_Contact( "General_Blend".Blend_Cluster2.CIP_Line1."CIP Request" )
      I_Contact( "General_Blend".Blend_Cluster2.CIP_Line2."CIP Request" )
      Coil( "General_Blend".Blend_Cluster2.CIP_Line3."CIP Enable" )
   END_RUNG
   // the same network as SCL:
   #_w1 := "AlwaysTRUE" AND NOT "Blend_T-31".Out_CIP_Req AND NOT "Blend_T-40".Out_CIP_Req AND NOT "Blend_T-41".Out_CIP_Req;
   "General_Blend".Blend_Cluster2.CIP_Line1."CIP Enable" := #_w1 AND NOT "Blend_T-31".State."Transfer 1 On Progress" AND NOT "Blend_T-40".State."Transfer 1 On Progress" AND NOT "Blend_T-41".State."Transfer 1 On Progress" AND NOT "General_Blend".Blend_Cluster2.CIP_Line2."CIP Request" AND NOT "General_Blend".Blend_Cluster2.CIP_Line3."CIP Request";
   "General_Blend".Blend_Cluster2.CIP_Line2."CIP Enable" := #_w1 AND NOT "Blend_T-31".State."Transfer 2 On Progress" AND NOT "Blend_T-40".State."Transfer 2 On Progress" AND NOT "Blend_T-41".State."Transfer 2 On Progress" AND NOT "General_Blend".Blend_Cluster2.CIP_Line1."CIP Request" AND NOT "General_Blend".Blend_Cluster2.CIP_Line3."CIP Request";
   "General_Blend".Blend_Cluster2.CIP_Line3."CIP Enable" := #_w1 AND NOT "Blend_T-31".State."Transfer 3 On Progress" AND NOT "Blend_T-40".State."Transfer 3 On Progress" AND NOT "Blend_T-41".State."Transfer 3 On Progress" AND NOT "General_Blend".Blend_Cluster2.CIP_Line1."CIP Request" AND NOT "General_Blend".Blend_Cluster2.CIP_Line2."CIP Request";
END_REGION

REGION Network 145: CIP Line Blending Cluster 2 Request
   RUNG wire#powerrail
      Contact( "AlwaysTRUE" )
      wire#w1
      Contact( "General_Blend".Blend_Cluster2.CIP_Line1."CIP Enable" )
      Contact( "General_Blend".Blend_Cluster2.CIP_Line1."CIP Request" )
      Contact( "General Buffer"."CIP Enable".Cluster2_Line1 )
      wire#w2
      Coil( "Mix_to_CIP".CIP_Request."Blending Cluster 2".Blending_Cluster2_LineProduct_Request )
   END_RUNG
   RUNG wire#w1
      Contact( "General_Blend".Blend_Cluster2.CIP_Line2."CIP Enable" )
      Contact( "General_Blend".Blend_Cluster2.CIP_Line2."CIP Request" )
      Contact( "General Buffer"."CIP Enable".Cluster2_Line2 )
   END_RUNG wire#w2
   RUNG wire#w1
      Contact( "General_Blend".Blend_Cluster2.CIP_Line3."CIP Enable" )
      Contact( "General_Blend".Blend_Cluster2.CIP_Line3."CIP Request" )
      Contact( "General Buffer"."CIP Enable".Cluster2_Line3 )
   END_RUNG wire#w2
   // the same network as SCL:
   "Mix_to_CIP".CIP_Request."Blending Cluster 2".Blending_Cluster2_LineProduct_Request := "AlwaysTRUE" AND (("General_Blend".Blend_Cluster2.CIP_Line1."CIP Enable" AND "General_Blend".Blend_Cluster2.CIP_Line1."CIP Request" AND "General Buffer"."CIP Enable".Cluster2_Line1) OR ("General_Blend".Blend_Cluster2.CIP_Line2."CIP Enable" AND "General_Blend".Blend_Cluster2.CIP_Line2."CIP Request" AND "General Buffer"."CIP Enable".Cluster2_Line2) OR ("General_Blend".Blend_Cluster2.CIP_Line3."CIP Enable" AND "General_Blend".Blend_Cluster2.CIP_Line3."CIP Request" AND "General Buffer"."CIP Enable".Cluster2_Line3));
END_REGION

REGION Network 146: CIP Line Blending Cluster 2 Line OK
   RUNG wire#powerrail
      Contact( "AlwaysTRUE" )
      wire#w1
      Contact( "General_Blend".Blend_Cluster2.CIP_Line1."CIP Request" )
      Contact( "IO_Valve_Buffer_DB"."AV-32.11".FB_OPEN )
      Contact( "IO_Valve_Blend41_DB"."AV-41.12".FB_OPEN )
      wire#w2
      Contact( "IO_Valve_Blend41_DB"."AV-41.13".FB_OPEN )
      wire#w3
      Contact( "General Buffer"."CIP Line Open".Cluster2_Line1 )
      wire#w4
      Coil( "Mix_to_CIP".CIP_Line_OK."Blending Cluster 2".Blending_Cluster2_LineProduct_LineOK )
   END_RUNG
   RUNG wire#w2
      Contact( "IO_Valve_Blend41_DB"."AV-41.14".FB_OPEN )
   END_RUNG wire#w3
   RUNG wire#w1
      Contact( "General_Blend".Blend_Cluster2.CIP_Line2."CIP Request" )
      Contact( "IO_Valve_Buffer_DB"."AV-32.11".FB_OPEN )
      Contact( "IO_Valve_Blend41_DB"."AV-41.15".FB_OPEN )
      wire#w5
      Contact( "IO_Valve_Blend41_DB"."AV-41.16".FB_OPEN )
      wire#w6
      Contact( "General Buffer"."CIP Line Open".Cluster2_Line2 )
   END_RUNG wire#w4
   RUNG wire#w5
      Contact( "IO_Valve_Blend41_DB"."AV-41.17".FB_OPEN )
   END_RUNG wire#w6
   RUNG wire#w1
      Contact( "General_Blend".Blend_Cluster2.CIP_Line3."CIP Request" )
      Contact( "IO_Valve_Buffer_DB"."AV-32.11".FB_OPEN )
      Contact( "IO_Valve_Blend41_DB"."AV-41.18".FB_OPEN )
      wire#w7
      Contact( "IO_Valve_Blend41_DB"."AV-41.19".FB_OPEN )
      wire#w8
      Contact( "General Buffer"."CIP Line Open".Cluster2_Line3 )
   END_RUNG wire#w4
   RUNG wire#w7
      Contact( "IO_Valve_Blend41_DB"."AV-41.20".FB_OPEN )
   END_RUNG wire#w8
   // the same network as SCL:
   "Mix_to_CIP".CIP_Line_OK."Blending Cluster 2".Blending_Cluster2_LineProduct_LineOK := "AlwaysTRUE" AND (("General_Blend".Blend_Cluster2.CIP_Line1."CIP Request" AND "IO_Valve_Buffer_DB"."AV-32.11".FB_OPEN AND "IO_Valve_Blend41_DB"."AV-41.12".FB_OPEN AND ("IO_Valve_Blend41_DB"."AV-41.13".FB_OPEN OR "IO_Valve_Blend41_DB"."AV-41.14".FB_OPEN) AND "General Buffer"."CIP Line Open".Cluster2_Line1) OR ("General_Blend".Blend_Cluster2.CIP_Line2."CIP Request" AND "IO_Valve_Buffer_DB"."AV-32.11".FB_OPEN AND "IO_Valve_Blend41_DB"."AV-41.15".FB_OPEN AND ("IO_Valve_Blend41_DB"."AV-41.16".FB_OPEN OR "IO_Valve_Blend41_DB"."AV-41.17".FB_OPEN) AND "General Buffer"."CIP Line Open".Cluster2_Line2) OR ("General_Blend".Blend_Cluster2.CIP_Line3."CIP Request" AND "IO_Valve_Buffer_DB"."AV-32.11".FB_OPEN AND "IO_Valve_Blend41_DB"."AV-41.18".FB_OPEN AND ("IO_Valve_Blend41_DB"."AV-41.19".FB_OPEN OR "IO_Valve_Blend41_DB"."AV-41.20".FB_OPEN) AND "General Buffer"."CIP Line Open".Cluster2_Line3));
END_REGION

REGION Network 147: CIP Line Blending Cluster 2 Valve Cmd
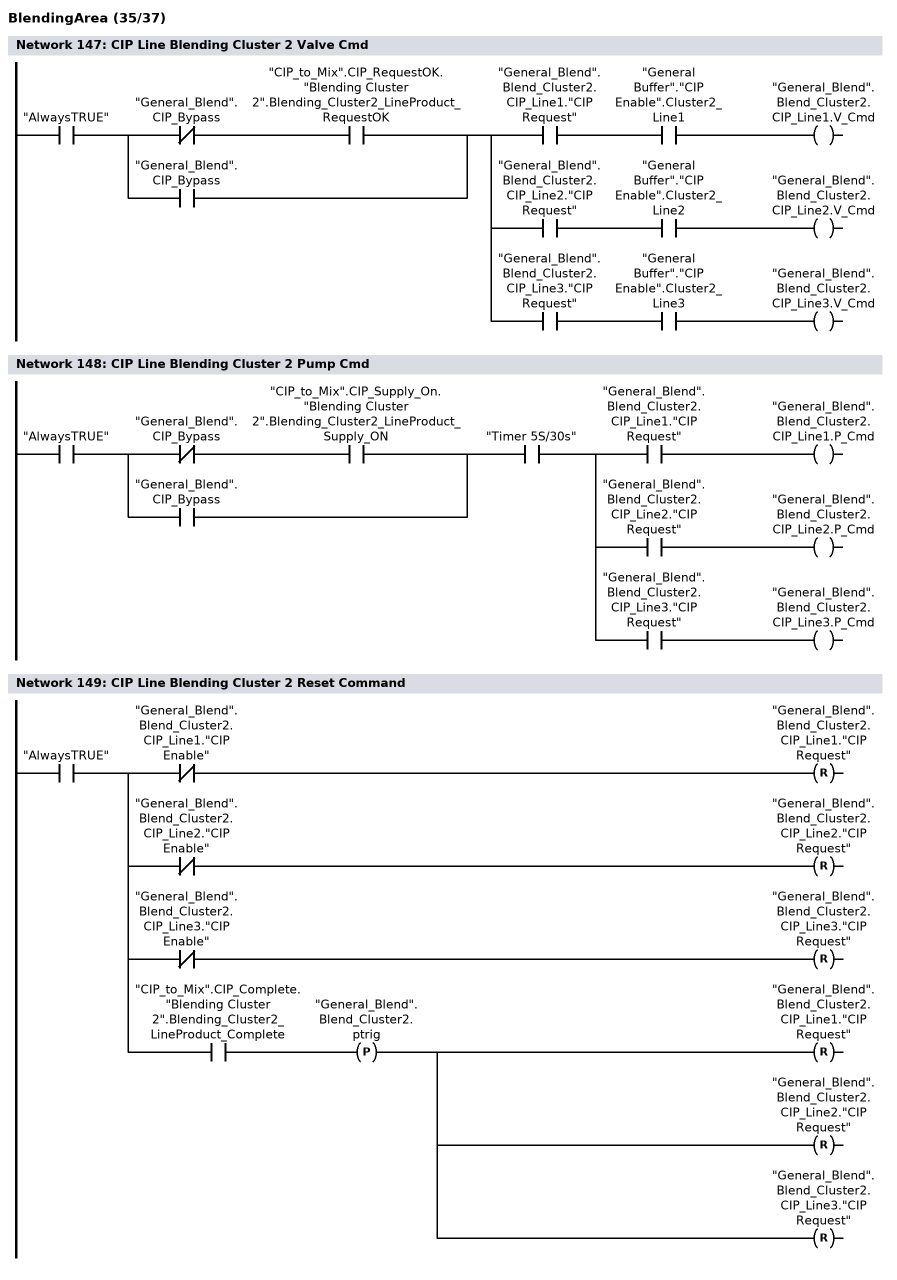
   RUNG wire#powerrail
      Contact( "AlwaysTRUE" )
      wire#w1
      I_Contact( "General_Blend".CIP_Bypass )
      Contact( "CIP_to_Mix".CIP_RequestOK."Blending Cluster 2".Blending_Cluster2_LineProduct_RequestOK )
      wire#w2
      Contact( "General_Blend".Blend_Cluster2.CIP_Line1."CIP Request" )
      Contact( "General Buffer"."CIP Enable".Cluster2_Line1 )
      Coil( "General_Blend".Blend_Cluster2.CIP_Line1.V_Cmd )
   END_RUNG
   RUNG wire#w1
      Contact( "General_Blend".CIP_Bypass )
   END_RUNG wire#w2
   RUNG wire#w2
      Contact( "General_Blend".Blend_Cluster2.CIP_Line2."CIP Request" )
      Contact( "General Buffer"."CIP Enable".Cluster2_Line2 )
      Coil( "General_Blend".Blend_Cluster2.CIP_Line2.V_Cmd )
   END_RUNG
   RUNG wire#w2
      Contact( "General_Blend".Blend_Cluster2.CIP_Line3."CIP Request" )
      Contact( "General Buffer"."CIP Enable".Cluster2_Line3 )
      Coil( "General_Blend".Blend_Cluster2.CIP_Line3.V_Cmd )
   END_RUNG
   // the same network as SCL:
   #_w1 := "AlwaysTRUE" AND ((NOT "General_Blend".CIP_Bypass AND "CIP_to_Mix".CIP_RequestOK."Blending Cluster 2".Blending_Cluster2_LineProduct_RequestOK) OR "General_Blend".CIP_Bypass);
   "General_Blend".Blend_Cluster2.CIP_Line1.V_Cmd := #_w1 AND "General_Blend".Blend_Cluster2.CIP_Line1."CIP Request" AND "General Buffer"."CIP Enable".Cluster2_Line1;
   "General_Blend".Blend_Cluster2.CIP_Line2.V_Cmd := #_w1 AND "General_Blend".Blend_Cluster2.CIP_Line2."CIP Request" AND "General Buffer"."CIP Enable".Cluster2_Line2;
   "General_Blend".Blend_Cluster2.CIP_Line3.V_Cmd := #_w1 AND "General_Blend".Blend_Cluster2.CIP_Line3."CIP Request" AND "General Buffer"."CIP Enable".Cluster2_Line3;
END_REGION

REGION Network 148: CIP Line Blending Cluster 2 Pump Cmd
   RUNG wire#powerrail
      Contact( "AlwaysTRUE" )
      wire#w1
      I_Contact( "General_Blend".CIP_Bypass )
      Contact( "CIP_to_Mix".CIP_Supply_On."Blending Cluster 2".Blending_Cluster2_LineProduct_Supply_ON )
      wire#w2
      Contact( "Timer 5S/30s" )
      wire#w3
      Contact( "General_Blend".Blend_Cluster2.CIP_Line1."CIP Request" )
      Coil( "General_Blend".Blend_Cluster2.CIP_Line1.P_Cmd )
   END_RUNG
   RUNG wire#w1
      Contact( "General_Blend".CIP_Bypass )
   END_RUNG wire#w2
   RUNG wire#w3
      Contact( "General_Blend".Blend_Cluster2.CIP_Line2."CIP Request" )
      Coil( "General_Blend".Blend_Cluster2.CIP_Line2.P_Cmd )
   END_RUNG
   RUNG wire#w3
      Contact( "General_Blend".Blend_Cluster2.CIP_Line3."CIP Request" )
      Coil( "General_Blend".Blend_Cluster2.CIP_Line3.P_Cmd )
   END_RUNG
   // the same network as SCL:
   #_w1 := "AlwaysTRUE" AND ((NOT "General_Blend".CIP_Bypass AND "CIP_to_Mix".CIP_Supply_On."Blending Cluster 2".Blending_Cluster2_LineProduct_Supply_ON) OR "General_Blend".CIP_Bypass) AND "Timer 5S/30s";
   "General_Blend".Blend_Cluster2.CIP_Line1.P_Cmd := #_w1 AND "General_Blend".Blend_Cluster2.CIP_Line1."CIP Request";
   "General_Blend".Blend_Cluster2.CIP_Line2.P_Cmd := #_w1 AND "General_Blend".Blend_Cluster2.CIP_Line2."CIP Request";
   "General_Blend".Blend_Cluster2.CIP_Line3.P_Cmd := #_w1 AND "General_Blend".Blend_Cluster2.CIP_Line3."CIP Request";
END_REGION

REGION Network 149: CIP Line Blending Cluster 2 Reset Command
   RUNG wire#powerrail
      Contact( "AlwaysTRUE" )
      wire#w1
      I_Contact( "General_Blend".Blend_Cluster2.CIP_Line1."CIP Enable" )
      R_Coil( "General_Blend".Blend_Cluster2.CIP_Line1."CIP Request" )
   END_RUNG
   RUNG wire#w1
      I_Contact( "General_Blend".Blend_Cluster2.CIP_Line2."CIP Enable" )
      R_Coil( "General_Blend".Blend_Cluster2.CIP_Line2."CIP Request" )
   END_RUNG
   RUNG wire#w1
      I_Contact( "General_Blend".Blend_Cluster2.CIP_Line3."CIP Enable" )
      R_Coil( "General_Blend".Blend_Cluster2.CIP_Line3."CIP Request" )
   END_RUNG
   RUNG wire#w1
      Contact( "CIP_to_Mix".CIP_Complete."Blending Cluster 2".Blending_Cluster2_LineProduct_Complete )
      P_Trig( "General_Blend".Blend_Cluster2.ptrig )
      wire#w2
      R_Coil( "General_Blend".Blend_Cluster2.CIP_Line1."CIP Request" )
   END_RUNG
   RUNG wire#w2
      R_Coil( "General_Blend".Blend_Cluster2.CIP_Line2."CIP Request" )
   END_RUNG
   RUNG wire#w2
      R_Coil( "General_Blend".Blend_Cluster2.CIP_Line3."CIP Request" )
   END_RUNG
   // the same network as SCL:
   IF "AlwaysTRUE" AND NOT "General_Blend".Blend_Cluster2.CIP_Line1."CIP Enable" THEN
       "General_Blend".Blend_Cluster2.CIP_Line1."CIP Request" := FALSE;
   END_IF;
   IF "AlwaysTRUE" AND NOT "General_Blend".Blend_Cluster2.CIP_Line2."CIP Enable" THEN
       "General_Blend".Blend_Cluster2.CIP_Line2."CIP Request" := FALSE;
   END_IF;
   IF "AlwaysTRUE" AND NOT "General_Blend".Blend_Cluster2.CIP_Line3."CIP Enable" THEN
       "General_Blend".Blend_Cluster2.CIP_Line3."CIP Request" := FALSE;
   END_IF;
   #_w1 := "AlwaysTRUE" AND "CIP_to_Mix".CIP_Complete."Blending Cluster 2".Blending_Cluster2_LineProduct_Complete;
   #_w2 := #_w1 AND NOT "General_Blend".Blend_Cluster2.ptrig;   // rising edge
   "General_Blend".Blend_Cluster2.ptrig := #_w1;
   IF #_w2 THEN
       "General_Blend".Blend_Cluster2.CIP_Line1."CIP Request" := FALSE;
       "General_Blend".Blend_Cluster2.CIP_Line2."CIP Request" := FALSE;
       "General_Blend".Blend_Cluster2.CIP_Line3."CIP Request" := FALSE;
   END_IF;
END_REGION

REGION Network 151: CIP to Return Line 1
   // Only for Blend Tank, Because CIP Supply from line 2 while Blend Tank can choose to return through line 1 or 2
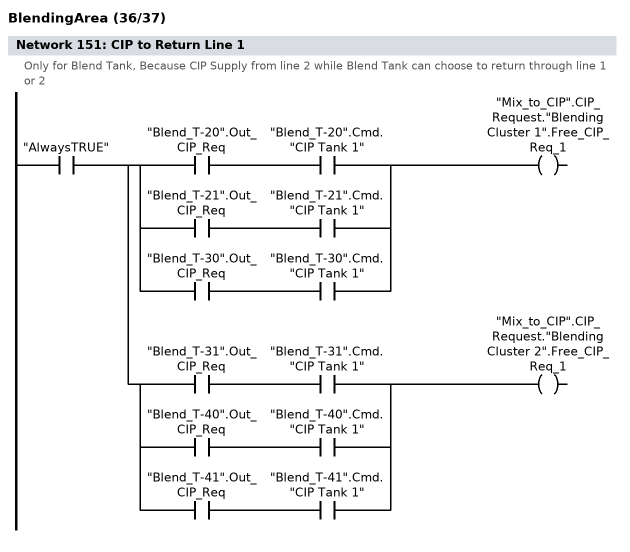
   RUNG wire#powerrail
      Contact( "AlwaysTRUE" )
      wire#w1
      Contact( "Blend_T-20".Out_CIP_Req )
      Contact( "Blend_T-20".Cmd."CIP Tank 1" )
      wire#w2
      Coil( "Mix_to_CIP".CIP_Request."Blending Cluster 1".Free_CIP_Req_1 )
   END_RUNG
   RUNG wire#w1
      Contact( "Blend_T-21".Out_CIP_Req )
      Contact( "Blend_T-21".Cmd."CIP Tank 1" )
   END_RUNG wire#w2
   RUNG wire#w1
      Contact( "Blend_T-30".Out_CIP_Req )
      Contact( "Blend_T-30".Cmd."CIP Tank 1" )
   END_RUNG wire#w2
   RUNG wire#w1
      Contact( "Blend_T-31".Out_CIP_Req )
      Contact( "Blend_T-31".Cmd."CIP Tank 1" )
      wire#w3
      Coil( "Mix_to_CIP".CIP_Request."Blending Cluster 2".Free_CIP_Req_1 )
   END_RUNG
   RUNG wire#w1
      Contact( "Blend_T-40".Out_CIP_Req )
      Contact( "Blend_T-40".Cmd."CIP Tank 1" )
   END_RUNG wire#w3
   RUNG wire#w1
      Contact( "Blend_T-41".Out_CIP_Req )
      Contact( "Blend_T-41".Cmd."CIP Tank 1" )
   END_RUNG wire#w3
   // the same network as SCL:
   "Mix_to_CIP".CIP_Request."Blending Cluster 1".Free_CIP_Req_1 := "AlwaysTRUE" AND (("Blend_T-20".Out_CIP_Req AND "Blend_T-20".Cmd."CIP Tank 1") OR ("Blend_T-21".Out_CIP_Req AND "Blend_T-21".Cmd."CIP Tank 1") OR ("Blend_T-30".Out_CIP_Req AND "Blend_T-30".Cmd."CIP Tank 1"));
   "Mix_to_CIP".CIP_Request."Blending Cluster 2".Free_CIP_Req_1 := "AlwaysTRUE" AND (("Blend_T-31".Out_CIP_Req AND "Blend_T-31".Cmd."CIP Tank 1") OR ("Blend_T-40".Out_CIP_Req AND "Blend_T-40".Cmd."CIP Tank 1") OR ("Blend_T-41".Out_CIP_Req AND "Blend_T-41".Cmd."CIP Tank 1"));
END_REGION

REGION Network 153: Valve
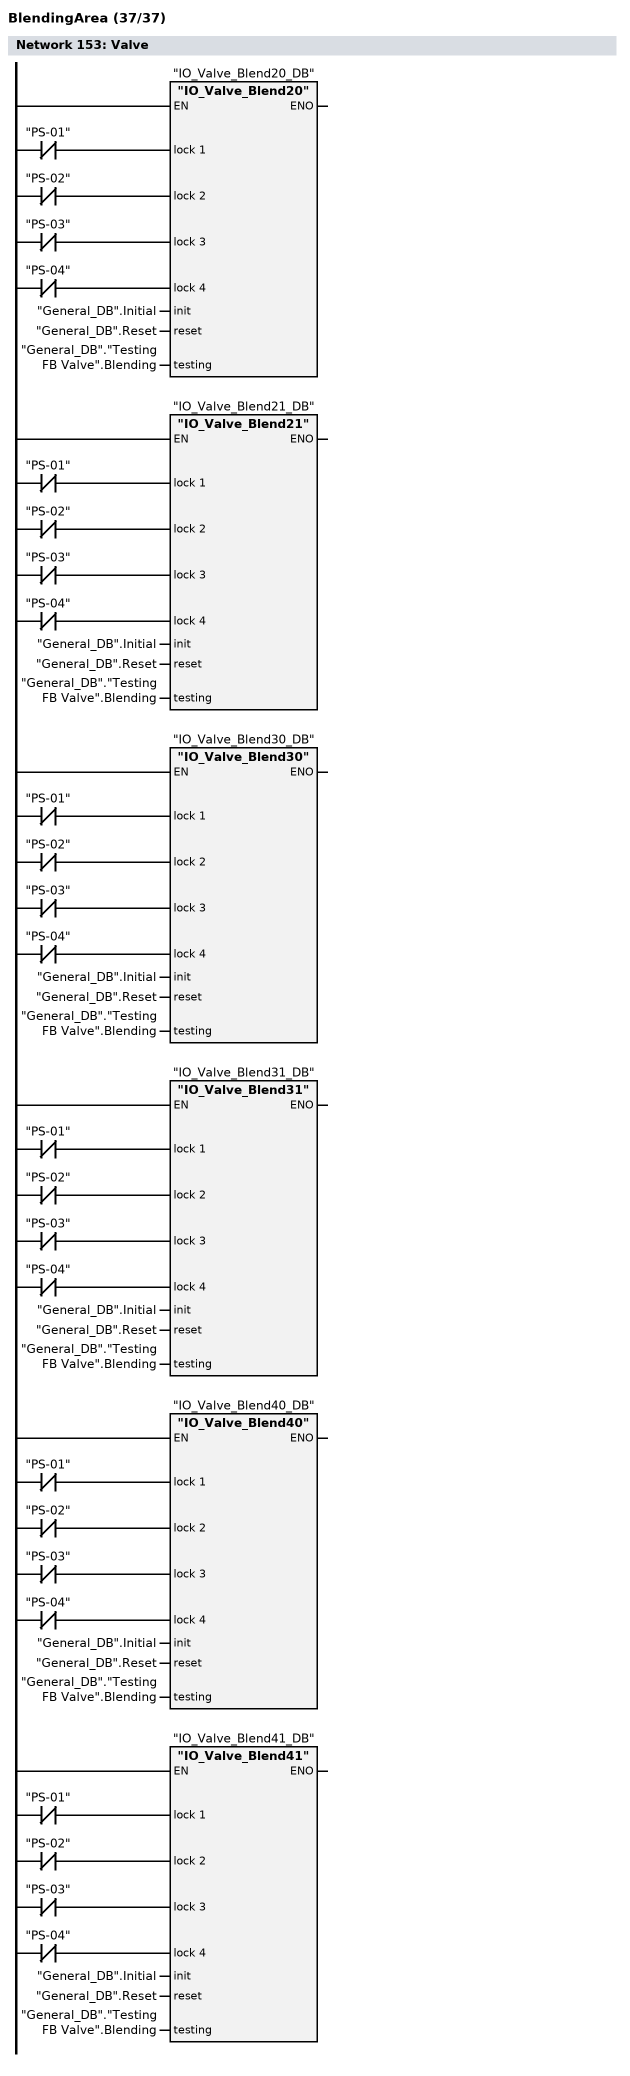
   RUNG wire#powerrail
      "IO_Valve_Blend20_DB"("lock 1" := wire#w1, "lock 2" := wire#w2, "lock 3" := wire#w3, "lock 4" := wire#w4, init := "General_DB".Initial, reset := "General_DB".Reset, testing := "General_DB"."Testing FB Valve".Blending)
   END_RUNG
   RUNG wire#powerrail
      I_Contact( "PS-01" )
   END_RUNG wire#w1
   RUNG wire#powerrail
      I_Contact( "PS-02" )
   END_RUNG wire#w2
   RUNG wire#powerrail
      I_Contact( "PS-03" )
   END_RUNG wire#w3
   RUNG wire#powerrail
      I_Contact( "PS-04" )
   END_RUNG wire#w4
   RUNG wire#powerrail
      "IO_Valve_Blend21_DB"("lock 1" := wire#w5, "lock 2" := wire#w6, "lock 3" := wire#w7, "lock 4" := wire#w8, init := "General_DB".Initial, reset := "General_DB".Reset, testing := "General_DB"."Testing FB Valve".Blending)
   END_RUNG
   RUNG wire#powerrail
      I_Contact( "PS-01" )
   END_RUNG wire#w5
   RUNG wire#powerrail
      I_Contact( "PS-02" )
   END_RUNG wire#w6
   RUNG wire#powerrail
      I_Contact( "PS-03" )
   END_RUNG wire#w7
   RUNG wire#powerrail
      I_Contact( "PS-04" )
   END_RUNG wire#w8
   RUNG wire#powerrail
      "IO_Valve_Blend30_DB"("lock 1" := wire#w9, "lock 2" := wire#w10, "lock 3" := wire#w11, "lock 4" := wire#w12, init := "General_DB".Initial, reset := "General_DB".Reset, testing := "General_DB"."Testing FB Valve".Blending)
   END_RUNG
   RUNG wire#powerrail
      I_Contact( "PS-01" )
   END_RUNG wire#w9
   RUNG wire#powerrail
      I_Contact( "PS-02" )
   END_RUNG wire#w10
   RUNG wire#powerrail
      I_Contact( "PS-03" )
   END_RUNG wire#w11
   RUNG wire#powerrail
      I_Contact( "PS-04" )
   END_RUNG wire#w12
   RUNG wire#powerrail
      "IO_Valve_Blend31_DB"("lock 1" := wire#w13, "lock 2" := wire#w14, "lock 3" := wire#w15, "lock 4" := wire#w16, init := "General_DB".Initial, reset := "General_DB".Reset, testing := "General_DB"."Testing FB Valve".Blending)
   END_RUNG
   RUNG wire#powerrail
      I_Contact( "PS-01" )
   END_RUNG wire#w13
   RUNG wire#powerrail
      I_Contact( "PS-02" )
   END_RUNG wire#w14
   RUNG wire#powerrail
      I_Contact( "PS-03" )
   END_RUNG wire#w15
   RUNG wire#powerrail
      I_Contact( "PS-04" )
   END_RUNG wire#w16
   RUNG wire#powerrail
      "IO_Valve_Blend40_DB"("lock 1" := wire#w17, "lock 2" := wire#w18, "lock 3" := wire#w19, "lock 4" := wire#w20, init := "General_DB".Initial, reset := "General_DB".Reset, testing := "General_DB"."Testing FB Valve".Blending)
   END_RUNG
   RUNG wire#powerrail
      I_Contact( "PS-01" )
   END_RUNG wire#w17
   RUNG wire#powerrail
      I_Contact( "PS-02" )
   END_RUNG wire#w18
   RUNG wire#powerrail
      I_Contact( "PS-03" )
   END_RUNG wire#w19
   RUNG wire#powerrail
      I_Contact( "PS-04" )
   END_RUNG wire#w20
   RUNG wire#powerrail
      "IO_Valve_Blend41_DB"("lock 1" := wire#w21, "lock 2" := wire#w22, "lock 3" := wire#w23, "lock 4" := wire#w24, init := "General_DB".Initial, reset := "General_DB".Reset, testing := "General_DB"."Testing FB Valve".Blending)
   END_RUNG
   RUNG wire#powerrail
      I_Contact( "PS-01" )
   END_RUNG wire#w21
   RUNG wire#powerrail
      I_Contact( "PS-02" )
   END_RUNG wire#w22
   RUNG wire#powerrail
      I_Contact( "PS-03" )
   END_RUNG wire#w23
   RUNG wire#powerrail
      I_Contact( "PS-04" )
   END_RUNG wire#w24
   // the same network as SCL:
   "IO_Valve_Blend20_DB"("lock 1" := NOT "PS-01",   // "IO_Valve_Blend20"
                         "lock 2" := NOT "PS-02",
                         "lock 3" := NOT "PS-03",
                         "lock 4" := NOT "PS-04",
                         init := "General_DB".Initial,
                         reset := "General_DB".Reset,
                         testing := "General_DB"."Testing FB Valve".Blending);
   "IO_Valve_Blend21_DB"("lock 1" := NOT "PS-01",   // "IO_Valve_Blend21"
                         "lock 2" := NOT "PS-02",
                         "lock 3" := NOT "PS-03",
                         "lock 4" := NOT "PS-04",
                         init := "General_DB".Initial,
                         reset := "General_DB".Reset,
                         testing := "General_DB"."Testing FB Valve".Blending);
   "IO_Valve_Blend30_DB"("lock 1" := NOT "PS-01",   // "IO_Valve_Blend30"
                         "lock 2" := NOT "PS-02",
                         "lock 3" := NOT "PS-03",
                         "lock 4" := NOT "PS-04",
                         init := "General_DB".Initial,
                         reset := "General_DB".Reset,
                         testing := "General_DB"."Testing FB Valve".Blending);
   "IO_Valve_Blend31_DB"("lock 1" := NOT "PS-01",   // "IO_Valve_Blend31"
                         "lock 2" := NOT "PS-02",
                         "lock 3" := NOT "PS-03",
                         "lock 4" := NOT "PS-04",
                         init := "General_DB".Initial,
                         reset := "General_DB".Reset,
                         testing := "General_DB"."Testing FB Valve".Blending);
   "IO_Valve_Blend40_DB"("lock 1" := NOT "PS-01",   // "IO_Valve_Blend40"
                         "lock 2" := NOT "PS-02",
                         "lock 3" := NOT "PS-03",
                         "lock 4" := NOT "PS-04",
                         init := "General_DB".Initial,
                         reset := "General_DB".Reset,
                         testing := "General_DB"."Testing FB Valve".Blending);
   "IO_Valve_Blend41_DB"("lock 1" := NOT "PS-01",   // "IO_Valve_Blend41"
                         "lock 2" := NOT "PS-02",
                         "lock 3" := NOT "PS-03",
                         "lock 4" := NOT "PS-04",
                         init := "General_DB".Initial,
                         reset := "General_DB".Reset,
                         testing := "General_DB"."Testing FB Valve".Blending);
END_REGION
END_FUNCTION

FUNCTION_BLOCK "IO Analog Blending"   // FB10, LAD
{ S7_Optimized_Access := 'FALSE' }
VERSION : 0.1
// stored: AutoNumber true, IsIECCheckEnabled false, SetENOAutomatically false, UDAEnableTagReadback false
   VAR_INPUT
      Init : Bool;
      Reset : Bool;
   END_VAR
   VAR
      "LT-20.01" { S7_SetPoint := 'True'} : "Ana_w_K1K2";
      "LT-21.01" { S7_SetPoint := 'True'} : "Ana_w_K1K2";
      "LT-22.01" { S7_SetPoint := 'True'} : "Ana_w_K1K2";
      "LT-30.01" { S7_SetPoint := 'True'} : "Ana_w_K1K2";
      "LT-31.01" { S7_SetPoint := 'True'} : "Ana_w_K1K2";
      "LT-32.01" { S7_SetPoint := 'True'} : "Ana_w_K1K2";
      "FT-15.01" { S7_SetPoint := 'True'} : "Ana_w_K1K2";
      "FT-15.01Com" { S7_SetPoint := 'True'} : "Read FT Comm";
      "FT-22.01" { S7_SetPoint := 'True'} : "Ana_w_K1K2";
      "FT-22.01Com" { S7_SetPoint := 'True'} : "Read FT Comm";
      "FT-32.01" { S7_SetPoint := 'True'} : "Ana_w_K1K2";
      "FT-32.01Com" { S7_SetPoint := 'True'} : "Read FT Comm";
      "LT-40.01" { S7_SetPoint := 'True'} : "Ana_w_K1K2";
      "LT-41.01" { S7_SetPoint := 'True'} : "Ana_w_K1K2";
      "FT-00.01" { S7_SetPoint := 'True'} : "Ana_w_K1K2";
   END_VAR
BEGIN

REGION Network 1: LT-20.01
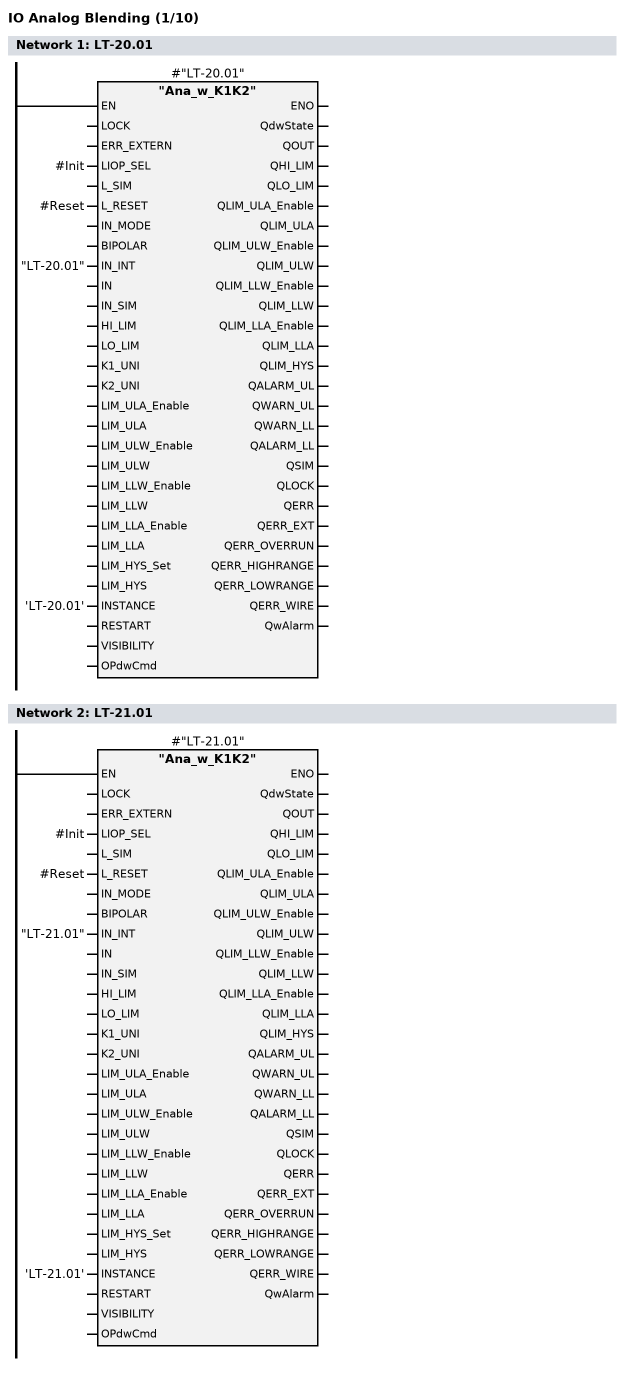
   RUNG wire#powerrail
      #"LT-20.01"(LOCK :=, ERR_EXTERN :=, LIOP_SEL := #Init, L_SIM :=, L_RESET := #Reset, IN_MODE :=, BIPOLAR :=, IN_INT := "LT-20.01", IN :=, IN_SIM :=, HI_LIM :=, LO_LIM :=, K1_UNI :=, K2_UNI :=, LIM_ULA_Enable :=, LIM_ULA :=, LIM_ULW_Enable :=, LIM_ULW :=, LIM_LLW_Enable :=, LIM_LLW :=, LIM_LLA_Enable :=, LIM_LLA :=, LIM_HYS_Set :=, LIM_HYS :=, INSTANCE := 'LT-20.01', RESTART :=, VISIBILITY :=, OPdwCmd :=, QdwState =>, QOUT =>, QHI_LIM =>, QLO_LIM =>, QLIM_ULA_Enable =>, QLIM_ULA =>, QLIM_ULW_Enable =>, QLIM_ULW =>, QLIM_LLW_Enable =>, QLIM_LLW =>, QLIM_LLA_Enable =>, QLIM_LLA =>, QLIM_HYS =>, QALARM_UL =>, QWARN_UL =>, QWARN_LL =>, QALARM_LL =>, QSIM =>, QLOCK =>, QERR =>, QERR_EXT =>, QERR_OVERRUN =>, QERR_HIGHRANGE =>, QERR_LOWRANGE =>, QERR_WIRE =>, QwAlarm =>)
   END_RUNG
   // the same network as SCL:
   #"LT-20.01"(LIOP_SEL := #Init, L_RESET := #Reset, IN_INT := "LT-20.01", INSTANCE := 'LT-20.01');   // "Ana_w_K1K2"
END_REGION

REGION Network 2: LT-21.01
   RUNG wire#powerrail
      #"LT-21.01"(LOCK :=, ERR_EXTERN :=, LIOP_SEL := #Init, L_SIM :=, L_RESET := #Reset, IN_MODE :=, BIPOLAR :=, IN_INT := "LT-21.01", IN :=, IN_SIM :=, HI_LIM :=, LO_LIM :=, K1_UNI :=, K2_UNI :=, LIM_ULA_Enable :=, LIM_ULA :=, LIM_ULW_Enable :=, LIM_ULW :=, LIM_LLW_Enable :=, LIM_LLW :=, LIM_LLA_Enable :=, LIM_LLA :=, LIM_HYS_Set :=, LIM_HYS :=, INSTANCE := 'LT-21.01', RESTART :=, VISIBILITY :=, OPdwCmd :=, QdwState =>, QOUT =>, QHI_LIM =>, QLO_LIM =>, QLIM_ULA_Enable =>, QLIM_ULA =>, QLIM_ULW_Enable =>, QLIM_ULW =>, QLIM_LLW_Enable =>, QLIM_LLW =>, QLIM_LLA_Enable =>, QLIM_LLA =>, QLIM_HYS =>, QALARM_UL =>, QWARN_UL =>, QWARN_LL =>, QALARM_LL =>, QSIM =>, QLOCK =>, QERR =>, QERR_EXT =>, QERR_OVERRUN =>, QERR_HIGHRANGE =>, QERR_LOWRANGE =>, QERR_WIRE =>, QwAlarm =>)
   END_RUNG
   // the same network as SCL:
   #"LT-21.01"(LIOP_SEL := #Init, L_RESET := #Reset, IN_INT := "LT-21.01", INSTANCE := 'LT-21.01');   // "Ana_w_K1K2"
END_REGION

REGION Network 3: LT-22.01
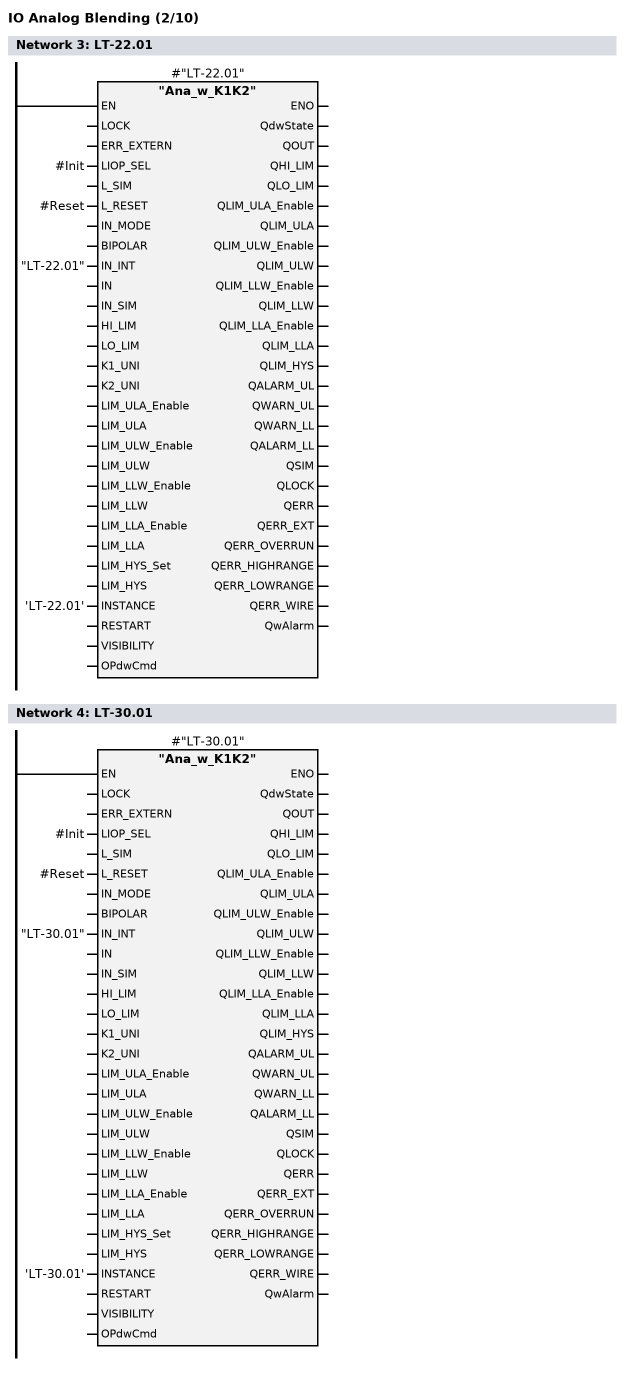
   RUNG wire#powerrail
      #"LT-22.01"(LOCK :=, ERR_EXTERN :=, LIOP_SEL := #Init, L_SIM :=, L_RESET := #Reset, IN_MODE :=, BIPOLAR :=, IN_INT := "LT-22.01", IN :=, IN_SIM :=, HI_LIM :=, LO_LIM :=, K1_UNI :=, K2_UNI :=, LIM_ULA_Enable :=, LIM_ULA :=, LIM_ULW_Enable :=, LIM_ULW :=, LIM_LLW_Enable :=, LIM_LLW :=, LIM_LLA_Enable :=, LIM_LLA :=, LIM_HYS_Set :=, LIM_HYS :=, INSTANCE := 'LT-22.01', RESTART :=, VISIBILITY :=, OPdwCmd :=, QdwState =>, QOUT =>, QHI_LIM =>, QLO_LIM =>, QLIM_ULA_Enable =>, QLIM_ULA =>, QLIM_ULW_Enable =>, QLIM_ULW =>, QLIM_LLW_Enable =>, QLIM_LLW =>, QLIM_LLA_Enable =>, QLIM_LLA =>, QLIM_HYS =>, QALARM_UL =>, QWARN_UL =>, QWARN_LL =>, QALARM_LL =>, QSIM =>, QLOCK =>, QERR =>, QERR_EXT =>, QERR_OVERRUN =>, QERR_HIGHRANGE =>, QERR_LOWRANGE =>, QERR_WIRE =>, QwAlarm =>)
   END_RUNG
   // the same network as SCL:
   #"LT-22.01"(LIOP_SEL := #Init, L_RESET := #Reset, IN_INT := "LT-22.01", INSTANCE := 'LT-22.01');   // "Ana_w_K1K2"
END_REGION

REGION Network 4: LT-30.01
   RUNG wire#powerrail
      #"LT-30.01"(LOCK :=, ERR_EXTERN :=, LIOP_SEL := #Init, L_SIM :=, L_RESET := #Reset, IN_MODE :=, BIPOLAR :=, IN_INT := "LT-30.01", IN :=, IN_SIM :=, HI_LIM :=, LO_LIM :=, K1_UNI :=, K2_UNI :=, LIM_ULA_Enable :=, LIM_ULA :=, LIM_ULW_Enable :=, LIM_ULW :=, LIM_LLW_Enable :=, LIM_LLW :=, LIM_LLA_Enable :=, LIM_LLA :=, LIM_HYS_Set :=, LIM_HYS :=, INSTANCE := 'LT-30.01', RESTART :=, VISIBILITY :=, OPdwCmd :=, QdwState =>, QOUT =>, QHI_LIM =>, QLO_LIM =>, QLIM_ULA_Enable =>, QLIM_ULA =>, QLIM_ULW_Enable =>, QLIM_ULW =>, QLIM_LLW_Enable =>, QLIM_LLW =>, QLIM_LLA_Enable =>, QLIM_LLA =>, QLIM_HYS =>, QALARM_UL =>, QWARN_UL =>, QWARN_LL =>, QALARM_LL =>, QSIM =>, QLOCK =>, QERR =>, QERR_EXT =>, QERR_OVERRUN =>, QERR_HIGHRANGE =>, QERR_LOWRANGE =>, QERR_WIRE =>, QwAlarm =>)
   END_RUNG
   // the same network as SCL:
   #"LT-30.01"(LIOP_SEL := #Init, L_RESET := #Reset, IN_INT := "LT-30.01", INSTANCE := 'LT-30.01');   // "Ana_w_K1K2"
END_REGION

REGION Network 5: LT-31.01
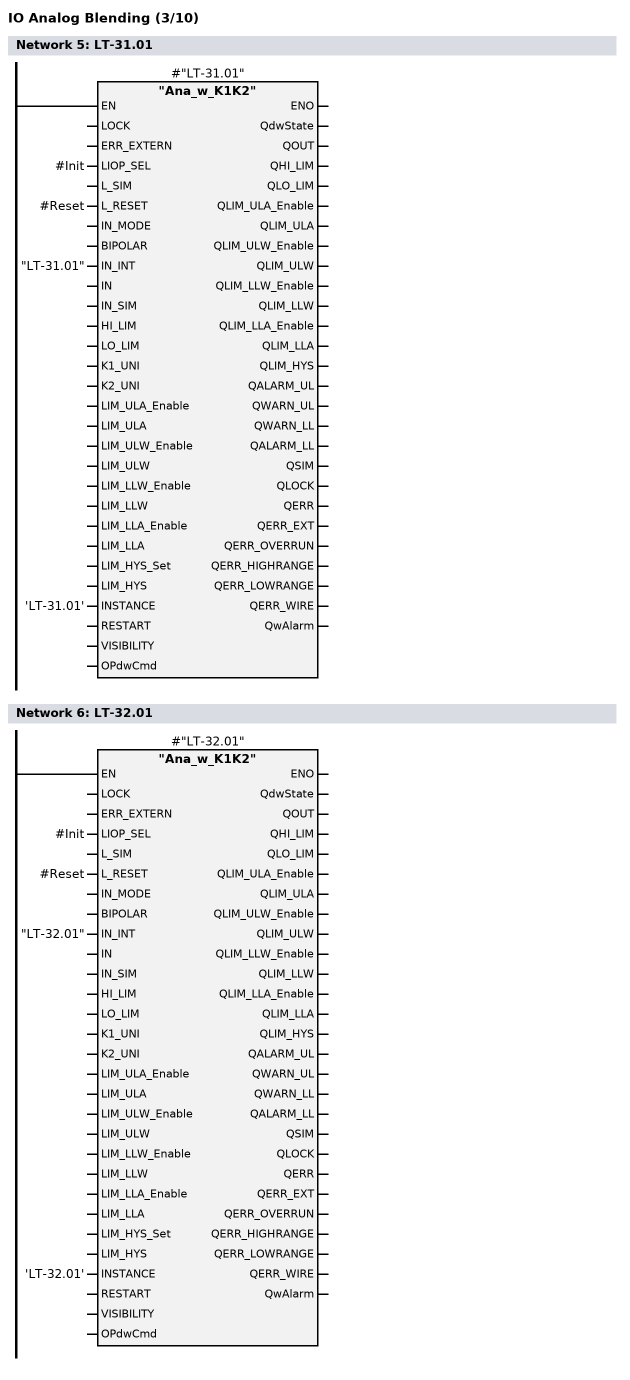
   RUNG wire#powerrail
      #"LT-31.01"(LOCK :=, ERR_EXTERN :=, LIOP_SEL := #Init, L_SIM :=, L_RESET := #Reset, IN_MODE :=, BIPOLAR :=, IN_INT := "LT-31.01", IN :=, IN_SIM :=, HI_LIM :=, LO_LIM :=, K1_UNI :=, K2_UNI :=, LIM_ULA_Enable :=, LIM_ULA :=, LIM_ULW_Enable :=, LIM_ULW :=, LIM_LLW_Enable :=, LIM_LLW :=, LIM_LLA_Enable :=, LIM_LLA :=, LIM_HYS_Set :=, LIM_HYS :=, INSTANCE := 'LT-31.01', RESTART :=, VISIBILITY :=, OPdwCmd :=, QdwState =>, QOUT =>, QHI_LIM =>, QLO_LIM =>, QLIM_ULA_Enable =>, QLIM_ULA =>, QLIM_ULW_Enable =>, QLIM_ULW =>, QLIM_LLW_Enable =>, QLIM_LLW =>, QLIM_LLA_Enable =>, QLIM_LLA =>, QLIM_HYS =>, QALARM_UL =>, QWARN_UL =>, QWARN_LL =>, QALARM_LL =>, QSIM =>, QLOCK =>, QERR =>, QERR_EXT =>, QERR_OVERRUN =>, QERR_HIGHRANGE =>, QERR_LOWRANGE =>, QERR_WIRE =>, QwAlarm =>)
   END_RUNG
   // the same network as SCL:
   #"LT-31.01"(LIOP_SEL := #Init, L_RESET := #Reset, IN_INT := "LT-31.01", INSTANCE := 'LT-31.01');   // "Ana_w_K1K2"
END_REGION

REGION Network 6: LT-32.01
   RUNG wire#powerrail
      #"LT-32.01"(LOCK :=, ERR_EXTERN :=, LIOP_SEL := #Init, L_SIM :=, L_RESET := #Reset, IN_MODE :=, BIPOLAR :=, IN_INT := "LT-32.01", IN :=, IN_SIM :=, HI_LIM :=, LO_LIM :=, K1_UNI :=, K2_UNI :=, LIM_ULA_Enable :=, LIM_ULA :=, LIM_ULW_Enable :=, LIM_ULW :=, LIM_LLW_Enable :=, LIM_LLW :=, LIM_LLA_Enable :=, LIM_LLA :=, LIM_HYS_Set :=, LIM_HYS :=, INSTANCE := 'LT-32.01', RESTART :=, VISIBILITY :=, OPdwCmd :=, QdwState =>, QOUT =>, QHI_LIM =>, QLO_LIM =>, QLIM_ULA_Enable =>, QLIM_ULA =>, QLIM_ULW_Enable =>, QLIM_ULW =>, QLIM_LLW_Enable =>, QLIM_LLW =>, QLIM_LLA_Enable =>, QLIM_LLA =>, QLIM_HYS =>, QALARM_UL =>, QWARN_UL =>, QWARN_LL =>, QALARM_LL =>, QSIM =>, QLOCK =>, QERR =>, QERR_EXT =>, QERR_OVERRUN =>, QERR_HIGHRANGE =>, QERR_LOWRANGE =>, QERR_WIRE =>, QwAlarm =>)
   END_RUNG
   // the same network as SCL:
   #"LT-32.01"(LIOP_SEL := #Init, L_RESET := #Reset, IN_INT := "LT-32.01", INSTANCE := 'LT-32.01');   // "Ana_w_K1K2"
END_REGION

REGION Network 7: LT-40.01
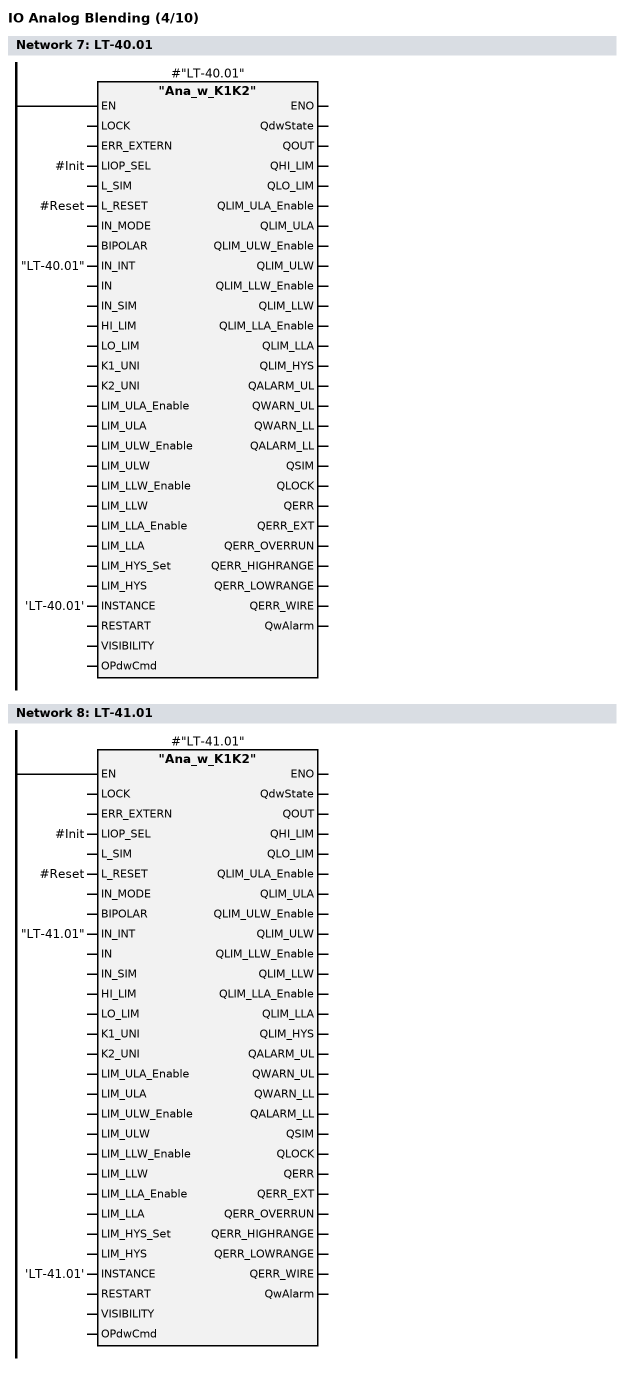
   RUNG wire#powerrail
      #"LT-40.01"(LOCK :=, ERR_EXTERN :=, LIOP_SEL := #Init, L_SIM :=, L_RESET := #Reset, IN_MODE :=, BIPOLAR :=, IN_INT := "LT-40.01", IN :=, IN_SIM :=, HI_LIM :=, LO_LIM :=, K1_UNI :=, K2_UNI :=, LIM_ULA_Enable :=, LIM_ULA :=, LIM_ULW_Enable :=, LIM_ULW :=, LIM_LLW_Enable :=, LIM_LLW :=, LIM_LLA_Enable :=, LIM_LLA :=, LIM_HYS_Set :=, LIM_HYS :=, INSTANCE := 'LT-40.01', RESTART :=, VISIBILITY :=, OPdwCmd :=, QdwState =>, QOUT =>, QHI_LIM =>, QLO_LIM =>, QLIM_ULA_Enable =>, QLIM_ULA =>, QLIM_ULW_Enable =>, QLIM_ULW =>, QLIM_LLW_Enable =>, QLIM_LLW =>, QLIM_LLA_Enable =>, QLIM_LLA =>, QLIM_HYS =>, QALARM_UL =>, QWARN_UL =>, QWARN_LL =>, QALARM_LL =>, QSIM =>, QLOCK =>, QERR =>, QERR_EXT =>, QERR_OVERRUN =>, QERR_HIGHRANGE =>, QERR_LOWRANGE =>, QERR_WIRE =>, QwAlarm =>)
   END_RUNG
   // the same network as SCL:
   #"LT-40.01"(LIOP_SEL := #Init, L_RESET := #Reset, IN_INT := "LT-40.01", INSTANCE := 'LT-40.01');   // "Ana_w_K1K2"
END_REGION

REGION Network 8: LT-41.01
   RUNG wire#powerrail
      #"LT-41.01"(LOCK :=, ERR_EXTERN :=, LIOP_SEL := #Init, L_SIM :=, L_RESET := #Reset, IN_MODE :=, BIPOLAR :=, IN_INT := "LT-41.01", IN :=, IN_SIM :=, HI_LIM :=, LO_LIM :=, K1_UNI :=, K2_UNI :=, LIM_ULA_Enable :=, LIM_ULA :=, LIM_ULW_Enable :=, LIM_ULW :=, LIM_LLW_Enable :=, LIM_LLW :=, LIM_LLA_Enable :=, LIM_LLA :=, LIM_HYS_Set :=, LIM_HYS :=, INSTANCE := 'LT-41.01', RESTART :=, VISIBILITY :=, OPdwCmd :=, QdwState =>, QOUT =>, QHI_LIM =>, QLO_LIM =>, QLIM_ULA_Enable =>, QLIM_ULA =>, QLIM_ULW_Enable =>, QLIM_ULW =>, QLIM_LLW_Enable =>, QLIM_LLW =>, QLIM_LLA_Enable =>, QLIM_LLA =>, QLIM_HYS =>, QALARM_UL =>, QWARN_UL =>, QWARN_LL =>, QALARM_LL =>, QSIM =>, QLOCK =>, QERR =>, QERR_EXT =>, QERR_OVERRUN =>, QERR_HIGHRANGE =>, QERR_LOWRANGE =>, QERR_WIRE =>, QwAlarm =>)
   END_RUNG
   // the same network as SCL:
   #"LT-41.01"(LIOP_SEL := #Init, L_RESET := #Reset, IN_INT := "LT-41.01", INSTANCE := 'LT-41.01');   // "Ana_w_K1K2"
END_REGION

REGION Network 9: FT-15.01 Communication
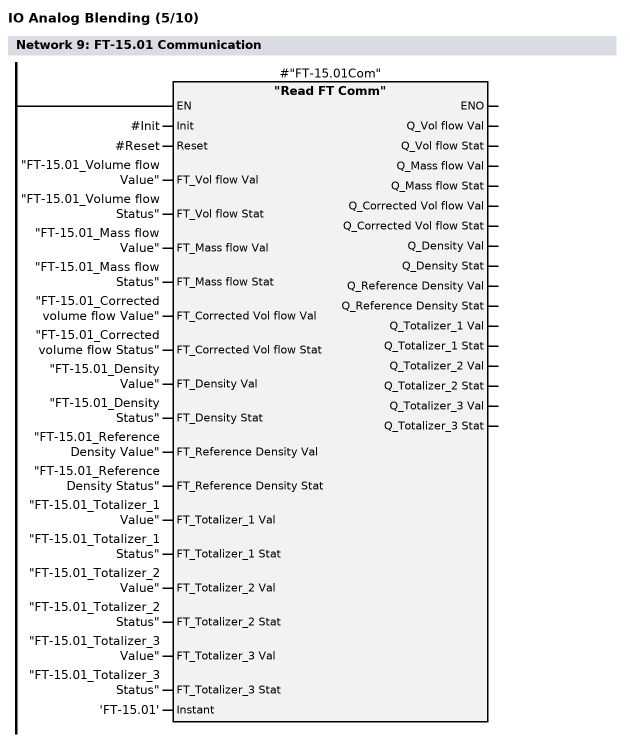
   RUNG wire#powerrail
      #"FT-15.01Com"(Init := #Init, Reset := #Reset, "FT_Vol flow Val" := "FT-15.01_Volume flow Value", "FT_Vol flow Stat" := "FT-15.01_Volume flow Status", "FT_Mass flow Val" := "FT-15.01_Mass flow Value", "FT_Mass flow Stat" := "FT-15.01_Mass flow Status", "FT_Corrected Vol flow Val" := "FT-15.01_Corrected volume flow Value", "FT_Corrected Vol flow Stat" := "FT-15.01_Corrected volume flow Status", "FT_Density Val" := "FT-15.01_Density Value", "FT_Density Stat" := "FT-15.01_Density Status", "FT_Reference Density Val" := "FT-15.01_Reference Density Value", "FT_Reference Density Stat" := "FT-15.01_Reference Density Status", "FT_Totalizer_1 Val" := "FT-15.01_Totalizer_1 Value", "FT_Totalizer_1 Stat" := "FT-15.01_Totalizer_1 Status", "FT_Totalizer_2 Val" := "FT-15.01_Totalizer_2 Value", "FT_Totalizer_2 Stat" := "FT-15.01_Totalizer_2 Status", "FT_Totalizer_3 Val" := "FT-15.01_Totalizer_3 Value", "FT_Totalizer_3 Stat" := "FT-15.01_Totalizer_3 Status", Instant := 'FT-15.01', "Q_Vol flow Val" =>, "Q_Vol flow Stat" =>, "Q_Mass flow Val" =>, "Q_Mass flow Stat" =>, "Q_Corrected Vol flow Val" =>, "Q_Corrected Vol flow Stat" =>, "Q_Density Val" =>, "Q_Density Stat" =>, "Q_Reference Density Val" =>, "Q_Reference Density Stat" =>, "Q_Totalizer_1 Val" =>, "Q_Totalizer_1 Stat" =>, "Q_Totalizer_2 Val" =>, "Q_Totalizer_2 Stat" =>, "Q_Totalizer_3 Val" =>, "Q_Totalizer_3 Stat" =>)
   END_RUNG
   // the same network as SCL:
   #"FT-15.01Com"(Init := #Init,   // "Read FT Comm"
                  Reset := #Reset,
                  "FT_Vol flow Val" := "FT-15.01_Volume flow Value",
                  "FT_Vol flow Stat" := "FT-15.01_Volume flow Status",
                  "FT_Mass flow Val" := "FT-15.01_Mass flow Value",
                  "FT_Mass flow Stat" := "FT-15.01_Mass flow Status",
                  "FT_Corrected Vol flow Val" := "FT-15.01_Corrected volume flow Value",
                  "FT_Corrected Vol flow Stat" := "FT-15.01_Corrected volume flow Status",
                  "FT_Density Val" := "FT-15.01_Density Value",
                  "FT_Density Stat" := "FT-15.01_Density Status",
                  "FT_Reference Density Val" := "FT-15.01_Reference Density Value",
                  "FT_Reference Density Stat" := "FT-15.01_Reference Density Status",
                  "FT_Totalizer_1 Val" := "FT-15.01_Totalizer_1 Value",
                  "FT_Totalizer_1 Stat" := "FT-15.01_Totalizer_1 Status",
                  "FT_Totalizer_2 Val" := "FT-15.01_Totalizer_2 Value",
                  "FT_Totalizer_2 Stat" := "FT-15.01_Totalizer_2 Status",
                  "FT_Totalizer_3 Val" := "FT-15.01_Totalizer_3 Value",
                  "FT_Totalizer_3 Stat" := "FT-15.01_Totalizer_3 Status",
                  Instant := 'FT-15.01');
END_REGION

REGION Network 10: FT-15.01 Flowrate
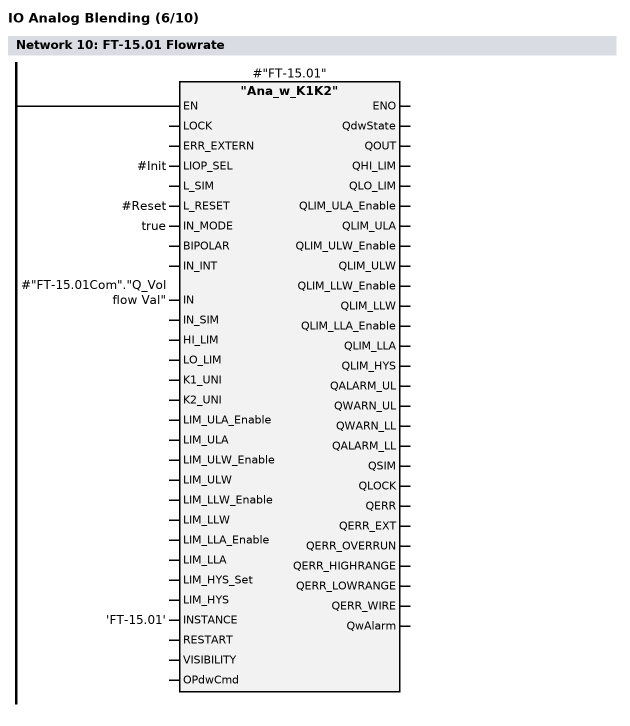
   RUNG wire#powerrail
      #"FT-15.01"(LOCK :=, ERR_EXTERN :=, LIOP_SEL := #Init, L_SIM :=, L_RESET := #Reset, IN_MODE := true, BIPOLAR :=, IN_INT :=, IN := #"FT-15.01Com"."Q_Vol flow Val", IN_SIM :=, HI_LIM :=, LO_LIM :=, K1_UNI :=, K2_UNI :=, LIM_ULA_Enable :=, LIM_ULA :=, LIM_ULW_Enable :=, LIM_ULW :=, LIM_LLW_Enable :=, LIM_LLW :=, LIM_LLA_Enable :=, LIM_LLA :=, LIM_HYS_Set :=, LIM_HYS :=, INSTANCE := 'FT-15.01', RESTART :=, VISIBILITY :=, OPdwCmd :=, QdwState =>, QOUT =>, QHI_LIM =>, QLO_LIM =>, QLIM_ULA_Enable =>, QLIM_ULA =>, QLIM_ULW_Enable =>, QLIM_ULW =>, QLIM_LLW_Enable =>, QLIM_LLW =>, QLIM_LLA_Enable =>, QLIM_LLA =>, QLIM_HYS =>, QALARM_UL =>, QWARN_UL =>, QWARN_LL =>, QALARM_LL =>, QSIM =>, QLOCK =>, QERR =>, QERR_EXT =>, QERR_OVERRUN =>, QERR_HIGHRANGE =>, QERR_LOWRANGE =>, QERR_WIRE =>, QwAlarm =>)
   END_RUNG
   // the same network as SCL:
   #"FT-15.01"(LIOP_SEL := #Init,   // "Ana_w_K1K2"
               L_RESET := #Reset,
               IN_MODE := true,
               IN := #"FT-15.01Com"."Q_Vol flow Val",
               INSTANCE := 'FT-15.01');
END_REGION

REGION Network 11: FT-22.01 Communication
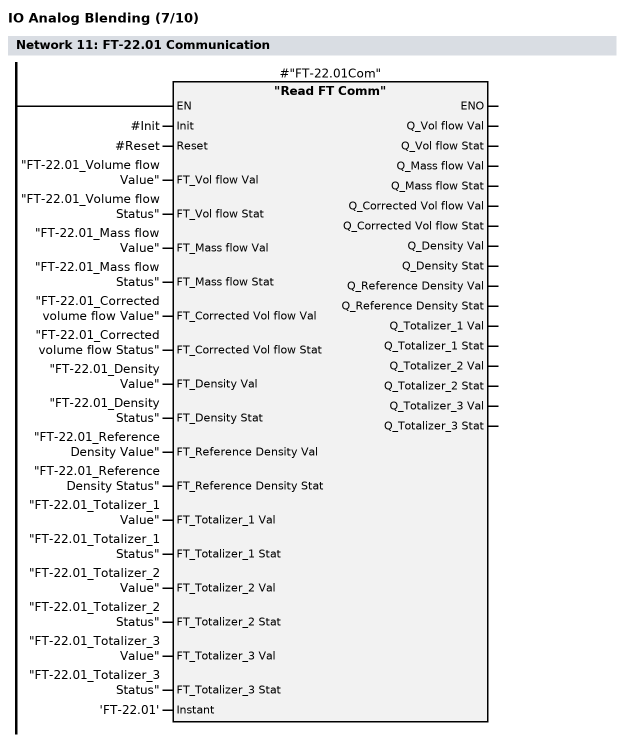
   RUNG wire#powerrail
      #"FT-22.01Com"(Init := #Init, Reset := #Reset, "FT_Vol flow Val" := "FT-22.01_Volume flow Value", "FT_Vol flow Stat" := "FT-22.01_Volume flow Status", "FT_Mass flow Val" := "FT-22.01_Mass flow Value", "FT_Mass flow Stat" := "FT-22.01_Mass flow Status", "FT_Corrected Vol flow Val" := "FT-22.01_Corrected volume flow Value", "FT_Corrected Vol flow Stat" := "FT-22.01_Corrected volume flow Status", "FT_Density Val" := "FT-22.01_Density Value", "FT_Density Stat" := "FT-22.01_Density Status", "FT_Reference Density Val" := "FT-22.01_Reference Density Value", "FT_Reference Density Stat" := "FT-22.01_Reference Density Status", "FT_Totalizer_1 Val" := "FT-22.01_Totalizer_1 Value", "FT_Totalizer_1 Stat" := "FT-22.01_Totalizer_1 Status", "FT_Totalizer_2 Val" := "FT-22.01_Totalizer_2 Value", "FT_Totalizer_2 Stat" := "FT-22.01_Totalizer_2 Status", "FT_Totalizer_3 Val" := "FT-22.01_Totalizer_3 Value", "FT_Totalizer_3 Stat" := "FT-22.01_Totalizer_3 Status", Instant := 'FT-22.01', "Q_Vol flow Val" =>, "Q_Vol flow Stat" =>, "Q_Mass flow Val" =>, "Q_Mass flow Stat" =>, "Q_Corrected Vol flow Val" =>, "Q_Corrected Vol flow Stat" =>, "Q_Density Val" =>, "Q_Density Stat" =>, "Q_Reference Density Val" =>, "Q_Reference Density Stat" =>, "Q_Totalizer_1 Val" =>, "Q_Totalizer_1 Stat" =>, "Q_Totalizer_2 Val" =>, "Q_Totalizer_2 Stat" =>, "Q_Totalizer_3 Val" =>, "Q_Totalizer_3 Stat" =>)
   END_RUNG
   // the same network as SCL:
   #"FT-22.01Com"(Init := #Init,   // "Read FT Comm"
                  Reset := #Reset,
                  "FT_Vol flow Val" := "FT-22.01_Volume flow Value",
                  "FT_Vol flow Stat" := "FT-22.01_Volume flow Status",
                  "FT_Mass flow Val" := "FT-22.01_Mass flow Value",
                  "FT_Mass flow Stat" := "FT-22.01_Mass flow Status",
                  "FT_Corrected Vol flow Val" := "FT-22.01_Corrected volume flow Value",
                  "FT_Corrected Vol flow Stat" := "FT-22.01_Corrected volume flow Status",
                  "FT_Density Val" := "FT-22.01_Density Value",
                  "FT_Density Stat" := "FT-22.01_Density Status",
                  "FT_Reference Density Val" := "FT-22.01_Reference Density Value",
                  "FT_Reference Density Stat" := "FT-22.01_Reference Density Status",
                  "FT_Totalizer_1 Val" := "FT-22.01_Totalizer_1 Value",
                  "FT_Totalizer_1 Stat" := "FT-22.01_Totalizer_1 Status",
                  "FT_Totalizer_2 Val" := "FT-22.01_Totalizer_2 Value",
                  "FT_Totalizer_2 Stat" := "FT-22.01_Totalizer_2 Status",
                  "FT_Totalizer_3 Val" := "FT-22.01_Totalizer_3 Value",
                  "FT_Totalizer_3 Stat" := "FT-22.01_Totalizer_3 Status",
                  Instant := 'FT-22.01');
END_REGION

REGION Network 12: FT-22.01 Flowrate
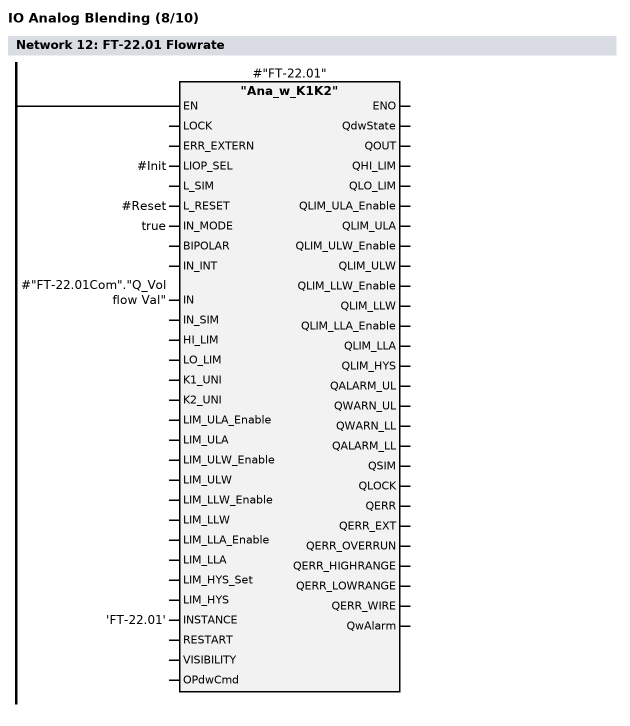
   RUNG wire#powerrail
      #"FT-22.01"(LOCK :=, ERR_EXTERN :=, LIOP_SEL := #Init, L_SIM :=, L_RESET := #Reset, IN_MODE := true, BIPOLAR :=, IN_INT :=, IN := #"FT-22.01Com"."Q_Vol flow Val", IN_SIM :=, HI_LIM :=, LO_LIM :=, K1_UNI :=, K2_UNI :=, LIM_ULA_Enable :=, LIM_ULA :=, LIM_ULW_Enable :=, LIM_ULW :=, LIM_LLW_Enable :=, LIM_LLW :=, LIM_LLA_Enable :=, LIM_LLA :=, LIM_HYS_Set :=, LIM_HYS :=, INSTANCE := 'FT-22.01', RESTART :=, VISIBILITY :=, OPdwCmd :=, QdwState =>, QOUT =>, QHI_LIM =>, QLO_LIM =>, QLIM_ULA_Enable =>, QLIM_ULA =>, QLIM_ULW_Enable =>, QLIM_ULW =>, QLIM_LLW_Enable =>, QLIM_LLW =>, QLIM_LLA_Enable =>, QLIM_LLA =>, QLIM_HYS =>, QALARM_UL =>, QWARN_UL =>, QWARN_LL =>, QALARM_LL =>, QSIM =>, QLOCK =>, QERR =>, QERR_EXT =>, QERR_OVERRUN =>, QERR_HIGHRANGE =>, QERR_LOWRANGE =>, QERR_WIRE =>, QwAlarm =>)
   END_RUNG
   // the same network as SCL:
   #"FT-22.01"(LIOP_SEL := #Init,   // "Ana_w_K1K2"
               L_RESET := #Reset,
               IN_MODE := true,
               IN := #"FT-22.01Com"."Q_Vol flow Val",
               INSTANCE := 'FT-22.01');
END_REGION

REGION Network 13: FT-32.01 Communication
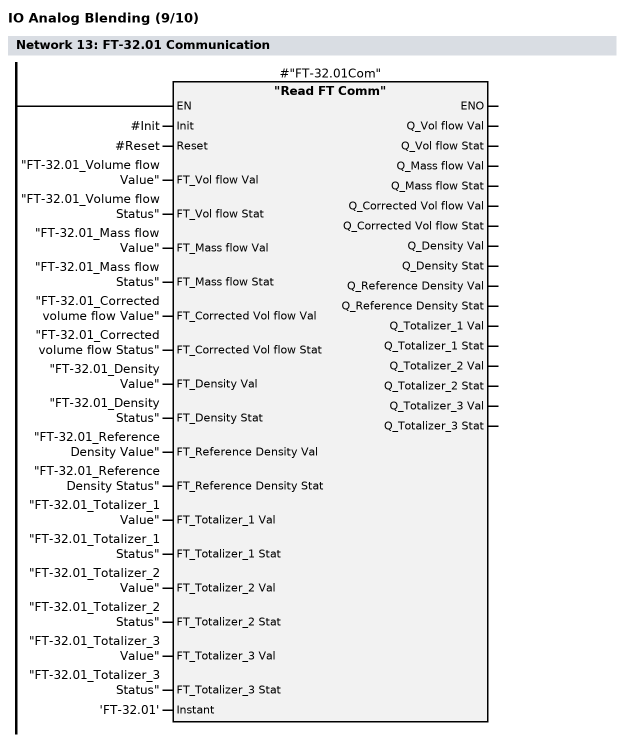
   RUNG wire#powerrail
      #"FT-32.01Com"(Init := #Init, Reset := #Reset, "FT_Vol flow Val" := "FT-32.01_Volume flow Value", "FT_Vol flow Stat" := "FT-32.01_Volume flow Status", "FT_Mass flow Val" := "FT-32.01_Mass flow Value", "FT_Mass flow Stat" := "FT-32.01_Mass flow Status", "FT_Corrected Vol flow Val" := "FT-32.01_Corrected volume flow Value", "FT_Corrected Vol flow Stat" := "FT-32.01_Corrected volume flow Status", "FT_Density Val" := "FT-32.01_Density Value", "FT_Density Stat" := "FT-32.01_Density Status", "FT_Reference Density Val" := "FT-32.01_Reference Density Value", "FT_Reference Density Stat" := "FT-32.01_Reference Density Status", "FT_Totalizer_1 Val" := "FT-32.01_Totalizer_1 Value", "FT_Totalizer_1 Stat" := "FT-32.01_Totalizer_1 Status", "FT_Totalizer_2 Val" := "FT-32.01_Totalizer_2 Value", "FT_Totalizer_2 Stat" := "FT-32.01_Totalizer_2 Status", "FT_Totalizer_3 Val" := "FT-32.01_Totalizer_3 Value", "FT_Totalizer_3 Stat" := "FT-32.01_Totalizer_3 Status", Instant := 'FT-32.01', "Q_Vol flow Val" =>, "Q_Vol flow Stat" =>, "Q_Mass flow Val" =>, "Q_Mass flow Stat" =>, "Q_Corrected Vol flow Val" =>, "Q_Corrected Vol flow Stat" =>, "Q_Density Val" =>, "Q_Density Stat" =>, "Q_Reference Density Val" =>, "Q_Reference Density Stat" =>, "Q_Totalizer_1 Val" =>, "Q_Totalizer_1 Stat" =>, "Q_Totalizer_2 Val" =>, "Q_Totalizer_2 Stat" =>, "Q_Totalizer_3 Val" =>, "Q_Totalizer_3 Stat" =>)
   END_RUNG
   // the same network as SCL:
   #"FT-32.01Com"(Init := #Init,   // "Read FT Comm"
                  Reset := #Reset,
                  "FT_Vol flow Val" := "FT-32.01_Volume flow Value",
                  "FT_Vol flow Stat" := "FT-32.01_Volume flow Status",
                  "FT_Mass flow Val" := "FT-32.01_Mass flow Value",
                  "FT_Mass flow Stat" := "FT-32.01_Mass flow Status",
                  "FT_Corrected Vol flow Val" := "FT-32.01_Corrected volume flow Value",
                  "FT_Corrected Vol flow Stat" := "FT-32.01_Corrected volume flow Status",
                  "FT_Density Val" := "FT-32.01_Density Value",
                  "FT_Density Stat" := "FT-32.01_Density Status",
                  "FT_Reference Density Val" := "FT-32.01_Reference Density Value",
                  "FT_Reference Density Stat" := "FT-32.01_Reference Density Status",
                  "FT_Totalizer_1 Val" := "FT-32.01_Totalizer_1 Value",
                  "FT_Totalizer_1 Stat" := "FT-32.01_Totalizer_1 Status",
                  "FT_Totalizer_2 Val" := "FT-32.01_Totalizer_2 Value",
                  "FT_Totalizer_2 Stat" := "FT-32.01_Totalizer_2 Status",
                  "FT_Totalizer_3 Val" := "FT-32.01_Totalizer_3 Value",
                  "FT_Totalizer_3 Stat" := "FT-32.01_Totalizer_3 Status",
                  Instant := 'FT-32.01');
END_REGION

REGION Network 14: FT-32.01 Flowrate
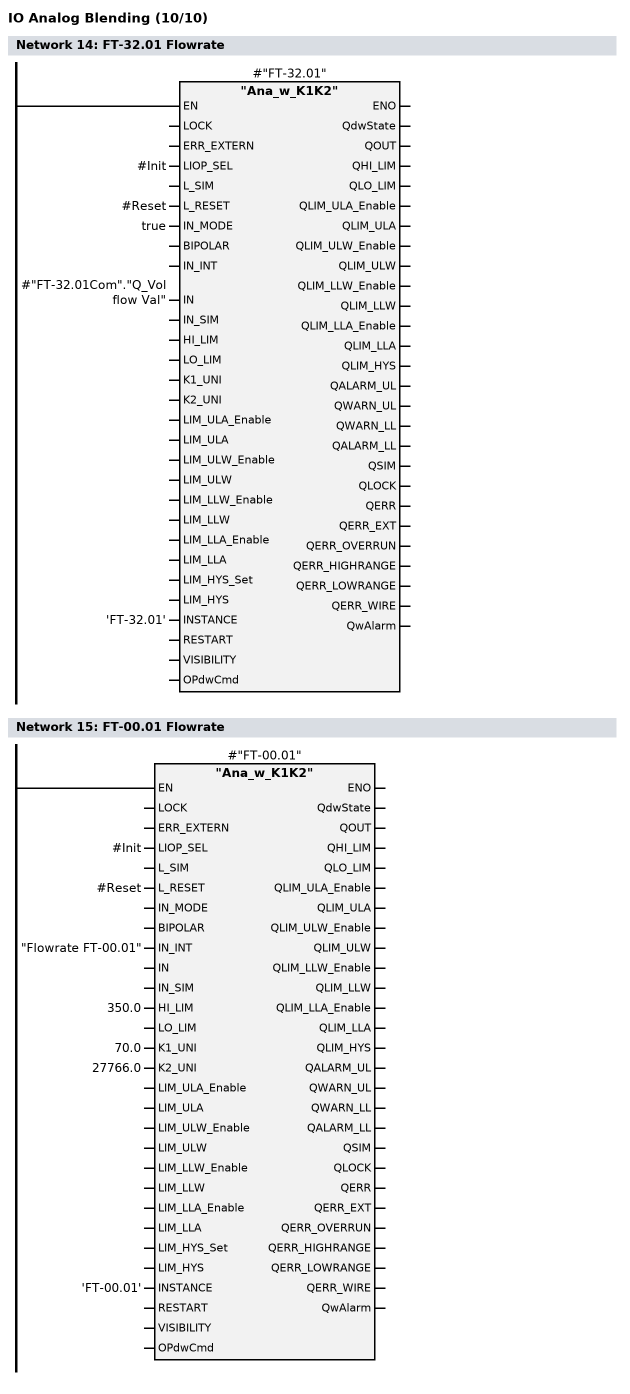
   RUNG wire#powerrail
      #"FT-32.01"(LOCK :=, ERR_EXTERN :=, LIOP_SEL := #Init, L_SIM :=, L_RESET := #Reset, IN_MODE := true, BIPOLAR :=, IN_INT :=, IN := #"FT-32.01Com"."Q_Vol flow Val", IN_SIM :=, HI_LIM :=, LO_LIM :=, K1_UNI :=, K2_UNI :=, LIM_ULA_Enable :=, LIM_ULA :=, LIM_ULW_Enable :=, LIM_ULW :=, LIM_LLW_Enable :=, LIM_LLW :=, LIM_LLA_Enable :=, LIM_LLA :=, LIM_HYS_Set :=, LIM_HYS :=, INSTANCE := 'FT-32.01', RESTART :=, VISIBILITY :=, OPdwCmd :=, QdwState =>, QOUT =>, QHI_LIM =>, QLO_LIM =>, QLIM_ULA_Enable =>, QLIM_ULA =>, QLIM_ULW_Enable =>, QLIM_ULW =>, QLIM_LLW_Enable =>, QLIM_LLW =>, QLIM_LLA_Enable =>, QLIM_LLA =>, QLIM_HYS =>, QALARM_UL =>, QWARN_UL =>, QWARN_LL =>, QALARM_LL =>, QSIM =>, QLOCK =>, QERR =>, QERR_EXT =>, QERR_OVERRUN =>, QERR_HIGHRANGE =>, QERR_LOWRANGE =>, QERR_WIRE =>, QwAlarm =>)
   END_RUNG
   // the same network as SCL:
   #"FT-32.01"(LIOP_SEL := #Init,   // "Ana_w_K1K2"
               L_RESET := #Reset,
               IN_MODE := true,
               IN := #"FT-32.01Com"."Q_Vol flow Val",
               INSTANCE := 'FT-32.01');
END_REGION

REGION Network 15: FT-00.01 Flowrate
   RUNG wire#powerrail
      #"FT-00.01"(LOCK :=, ERR_EXTERN :=, LIOP_SEL := #Init, L_SIM :=, L_RESET := #Reset, IN_MODE :=, BIPOLAR :=, IN_INT := "Flowrate FT-00.01", IN :=, IN_SIM :=, HI_LIM := 350.0, LO_LIM :=, K1_UNI := 70.0, K2_UNI := 27766.0, LIM_ULA_Enable :=, LIM_ULA :=, LIM_ULW_Enable :=, LIM_ULW :=, LIM_LLW_Enable :=, LIM_LLW :=, LIM_LLA_Enable :=, LIM_LLA :=, LIM_HYS_Set :=, LIM_HYS :=, INSTANCE := 'FT-00.01', RESTART :=, VISIBILITY :=, OPdwCmd :=, QdwState =>, QOUT =>, QHI_LIM =>, QLO_LIM =>, QLIM_ULA_Enable =>, QLIM_ULA =>, QLIM_ULW_Enable =>, QLIM_ULW =>, QLIM_LLW_Enable =>, QLIM_LLW =>, QLIM_LLA_Enable =>, QLIM_LLA =>, QLIM_HYS =>, QALARM_UL =>, QWARN_UL =>, QWARN_LL =>, QALARM_LL =>, QSIM =>, QLOCK =>, QERR =>, QERR_EXT =>, QERR_OVERRUN =>, QERR_HIGHRANGE =>, QERR_LOWRANGE =>, QERR_WIRE =>, QwAlarm =>)
   END_RUNG
   // the same network as SCL:
   #"FT-00.01"(LIOP_SEL := #Init,   // "Ana_w_K1K2"
               L_RESET := #Reset,
               IN_INT := "Flowrate FT-00.01",
               HI_LIM := 350.0,
               K1_UNI := 70.0,
               K2_UNI := 27766.0,
               INSTANCE := 'FT-00.01');
END_REGION
END_FUNCTION_BLOCK

FUNCTION_BLOCK "IO Digital Blending"   // FB6, LAD
{ S7_Optimized_Access := 'FALSE' }
VERSION : 0.1
// stored: AutoNumber true, IsIECCheckEnabled false, SetENOAutomatically false, UDAEnableTagReadback false
   VAR_INPUT
      Init : Bool;
      Reset : Bool;
   END_VAR
   VAR
      "DRP-P22.01" { S7_SetPoint := 'True'} : "Digital";   // DRY RUN PROTECTION MONO PUMP P-22.01
      "DRP-P32.01" { S7_SetPoint := 'True'} : "Digital";   // DRY RUN PROTECTION MONO PUMP P-32.01
   END_VAR
BEGIN

REGION Network 1: DRP-P22.01
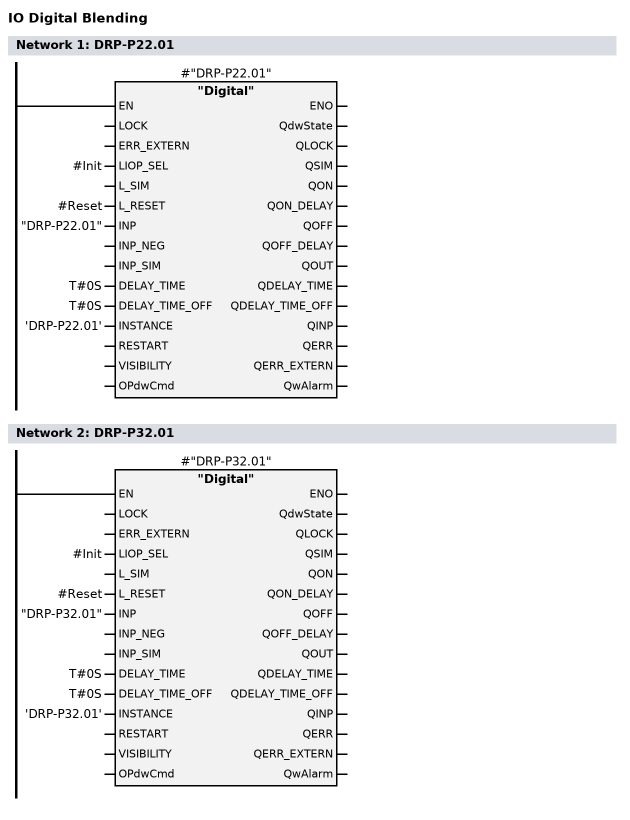
   RUNG wire#powerrail
      #"DRP-P22.01"(LOCK :=, ERR_EXTERN :=, LIOP_SEL := #Init, L_SIM :=, L_RESET := #Reset, INP := "DRP-P22.01", INP_NEG :=, INP_SIM :=, DELAY_TIME := T#0S, DELAY_TIME_OFF := T#0S, INSTANCE := 'DRP-P22.01', RESTART :=, VISIBILITY :=, OPdwCmd :=, QdwState =>, QLOCK =>, QSIM =>, QON =>, QON_DELAY =>, QOFF =>, QOFF_DELAY =>, QOUT =>, QDELAY_TIME =>, QDELAY_TIME_OFF =>, QINP =>, QERR =>, QERR_EXTERN =>, QwAlarm =>)
   END_RUNG
   // the same network as SCL:
   #"DRP-P22.01"(LIOP_SEL := #Init,   // "Digital"
                 L_RESET := #Reset,
                 INP := "DRP-P22.01",
                 DELAY_TIME := T#0S,
                 DELAY_TIME_OFF := T#0S,
                 INSTANCE := 'DRP-P22.01');
END_REGION

REGION Network 2: DRP-P32.01
   RUNG wire#powerrail
      #"DRP-P32.01"(LOCK :=, ERR_EXTERN :=, LIOP_SEL := #Init, L_SIM :=, L_RESET := #Reset, INP := "DRP-P32.01", INP_NEG :=, INP_SIM :=, DELAY_TIME := T#0S, DELAY_TIME_OFF := T#0S, INSTANCE := 'DRP-P32.01', RESTART :=, VISIBILITY :=, OPdwCmd :=, QdwState =>, QLOCK =>, QSIM =>, QON =>, QON_DELAY =>, QOFF =>, QOFF_DELAY =>, QOUT =>, QDELAY_TIME =>, QDELAY_TIME_OFF =>, QINP =>, QERR =>, QERR_EXTERN =>, QwAlarm =>)
   END_RUNG
   // the same network as SCL:
   #"DRP-P32.01"(LIOP_SEL := #Init,   // "Digital"
                 L_RESET := #Reset,
                 INP := "DRP-P32.01",
                 DELAY_TIME := T#0S,
                 DELAY_TIME_OFF := T#0S,
                 INSTANCE := 'DRP-P32.01');
END_REGION
END_FUNCTION_BLOCK

FUNCTION_BLOCK "Alarm Flow Collector"   // FB211, LAD
{ S7_Optimized_Access := 'TRUE' }
VERSION : 0.1
// stored: AutoNumber false, IsIECCheckEnabled false, IsRetainMemResEnabled false, MemoryReserve 100, SetENOAutomatically false, UDAEnableTagReadback false
   VAR_INPUT
      Reset : Bool;
   END_VAR
   VAR
      alwaysON : Bool;
   END_VAR
   VAR RETAIN
      Param : Struct
         min_Flow : Struct
            ChiliAwetan1 : Real := 5.0;
            ChiliAwetan2 : Real := 5.0;
            ChiliAwetan3 : Real := 5.0;
            Tomato : Real := 5.0;
            ChiliFresh1 : Real := 5.0;
            ChiliFresh2 : Real := 5.0;
            ChiliFresh3 : Real := 5.0;
            Garlic : Real := 5.0;
            HW : Real := 5.0;
            Vinegar : Real := 5.0;
            Sugar : Real := 5.0;
            Salt : Real := 5.0;
            ProWater : Real := 5.0;
            Homomixer : Real := 5.0;
         END_STRUCT;
         timerMon : Struct
            ChiliAwetan1 : TON_TIME;
            ChiliAwetan2 : TON_TIME;
            ChiliAwetan3 : TON_TIME;
            Tomato : TON_TIME;
            ChiliFresh1 : TON_TIME;
            ChiliFresh2 : TON_TIME;
            ChiliFresh3 : TON_TIME;
            Garlic : TON_TIME;
            HW : TON_TIME;
            Vinegar : TON_TIME;
            Sugar : TON_TIME;
            Salt : TON_TIME;
            ProWater : TON_TIME;
            Homomixer : TON_TIME;
         END_STRUCT;
      END_STRUCT;
   END_VAR
   VAR
      AlarmFlow_Blend : Word;
   END_VAR
   // Param.timerMon.ChiliAwetan1.PT := T#20s;
   // Param.timerMon.ChiliAwetan2.PT := T#20s;
   // Param.timerMon.ChiliAwetan3.PT := T#20s;
   // Param.timerMon.Tomato.PT := T#20s;
   // Param.timerMon.ChiliFresh1.PT := T#20s;
   // Param.timerMon.ChiliFresh2.PT := T#20s;
   // Param.timerMon.ChiliFresh3.PT := T#20s;
   // Param.timerMon.Garlic.PT := T#20s;
   // Param.timerMon.HW.PT := T#20s;
   // Param.timerMon.Vinegar.PT := T#20s;
   // Param.timerMon.Sugar.PT := T#20s;
   // Param.timerMon.Salt.PT := T#20s;
   // Param.timerMon.ProWater.PT := T#20s;
   // Param.timerMon.Homomixer.PT := T#20s;
BEGIN

REGION Network 1: always ON
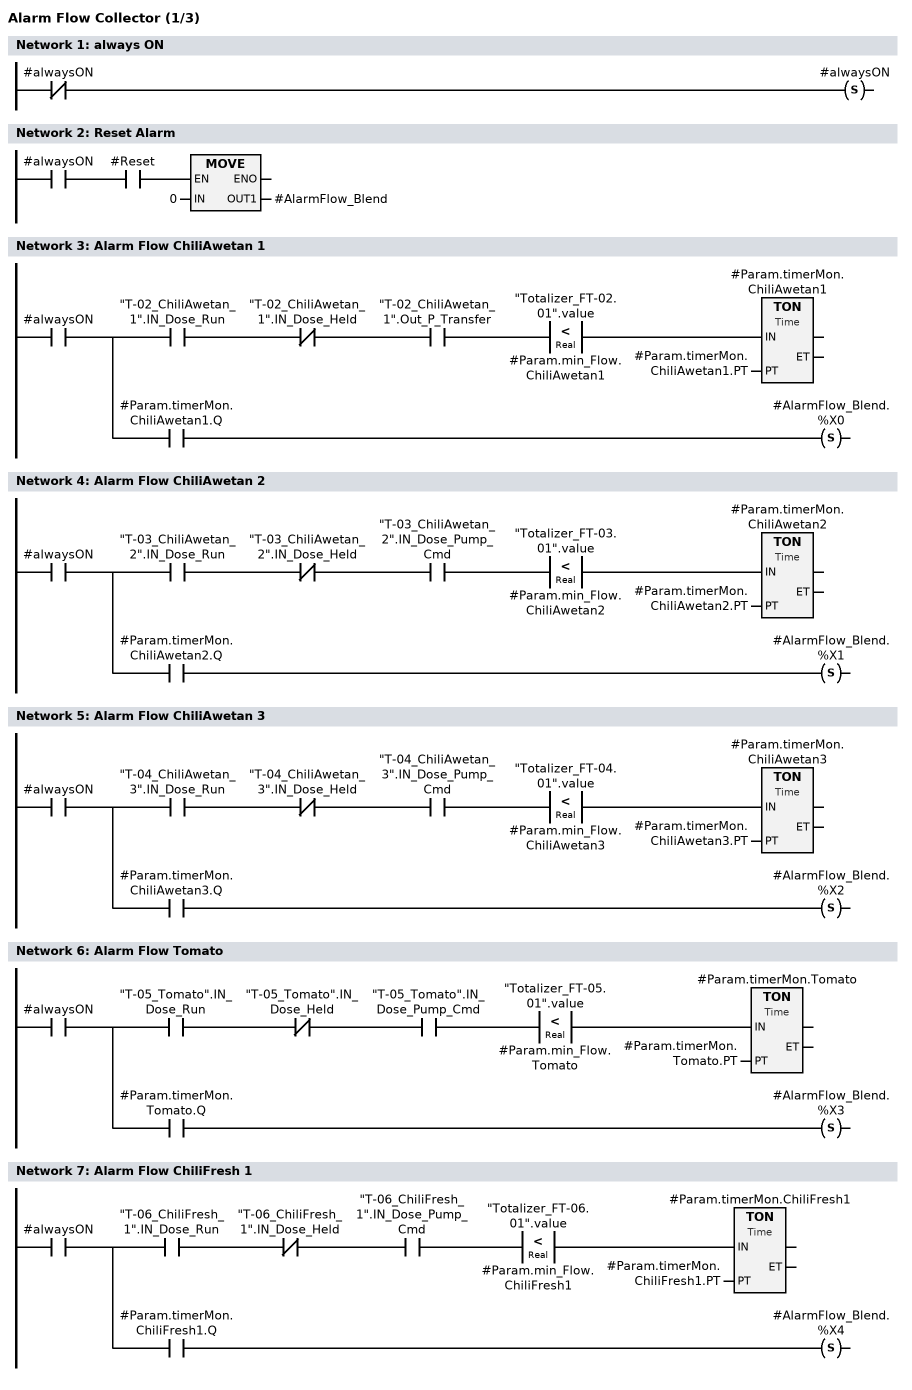
   RUNG wire#powerrail
      I_Contact( #alwaysON )
      S_Coil( #alwaysON )
   END_RUNG
   // the same network as SCL:
   IF NOT #alwaysON THEN #alwaysON := TRUE; END_IF;
END_REGION

REGION Network 2: Reset Alarm
   RUNG wire#powerrail
      Contact( #alwaysON )
      Contact( #Reset )
      Move(in := 0, out1 => #AlarmFlow_Blend)
   END_RUNG
   // the same network as SCL:
   IF #alwaysON AND #Reset THEN #AlarmFlow_Blend := 0; END_IF;
END_REGION

REGION Network 3: Alarm Flow ChiliAwetan 1
   RUNG wire#powerrail
      Contact( #alwaysON )
      wire#w1
      Contact( "T-02_ChiliAwetan_1".IN_Dose_Run )
      I_Contact( "T-02_ChiliAwetan_1".IN_Dose_Held )
      Contact( "T-02_ChiliAwetan_1".Out_P_Transfer )
      { S7_Templates := "SrcType := Real" } LT_Contact(in1 := "Totalizer_FT-02.01".value, in2 := #Param.min_Flow.ChiliAwetan1)
      { S7_Templates := "time_type := Time" } #Param.timerMon.ChiliAwetan1.TON(pt := #Param.timerMon.ChiliAwetan1.PT, et =>)
   END_RUNG
   RUNG wire#w1
      Contact( #Param.timerMon.ChiliAwetan1.Q )
      S_Coil( #AlarmFlow_Blend.%X0 )
   END_RUNG
   // the same network as SCL:
   #Param.timerMon.ChiliAwetan1.TON(IN := #alwaysON AND "T-02_ChiliAwetan_1".IN_Dose_Run AND NOT "T-02_ChiliAwetan_1".IN_Dose_Held AND "T-02_ChiliAwetan_1".Out_P_Transfer AND ("Totalizer_FT-02.01".value < #Param.min_Flow.ChiliAwetan1),
                           PT := #Param.timerMon.ChiliAwetan1.PT);
   IF #alwaysON AND #Param.timerMon.ChiliAwetan1.Q THEN #AlarmFlow_Blend.%X0 := TRUE; END_IF;
END_REGION

REGION Network 4: Alarm Flow ChiliAwetan 2
   RUNG wire#powerrail
      Contact( #alwaysON )
      wire#w1
      Contact( "T-03_ChiliAwetan_2".IN_Dose_Run )
      I_Contact( "T-03_ChiliAwetan_2".IN_Dose_Held )
      Contact( "T-03_ChiliAwetan_2".IN_Dose_Pump_Cmd )
      { S7_Templates := "SrcType := Real" } LT_Contact(in1 := "Totalizer_FT-03.01".value, in2 := #Param.min_Flow.ChiliAwetan2)
      { S7_Templates := "time_type := Time" } #Param.timerMon.ChiliAwetan2.TON(pt := #Param.timerMon.ChiliAwetan2.PT, et =>)
   END_RUNG
   RUNG wire#w1
      Contact( #Param.timerMon.ChiliAwetan2.Q )
      S_Coil( #AlarmFlow_Blend.%X1 )
   END_RUNG
   // the same network as SCL:
   #Param.timerMon.ChiliAwetan2.TON(IN := #alwaysON AND "T-03_ChiliAwetan_2".IN_Dose_Run AND NOT "T-03_ChiliAwetan_2".IN_Dose_Held AND "T-03_ChiliAwetan_2".IN_Dose_Pump_Cmd AND ("Totalizer_FT-03.01".value < #Param.min_Flow.ChiliAwetan2),
                           PT := #Param.timerMon.ChiliAwetan2.PT);
   IF #alwaysON AND #Param.timerMon.ChiliAwetan2.Q THEN #AlarmFlow_Blend.%X1 := TRUE; END_IF;
END_REGION

REGION Network 5: Alarm Flow ChiliAwetan 3
   RUNG wire#powerrail
      Contact( #alwaysON )
      wire#w1
      Contact( "T-04_ChiliAwetan_3".IN_Dose_Run )
      I_Contact( "T-04_ChiliAwetan_3".IN_Dose_Held )
      Contact( "T-04_ChiliAwetan_3".IN_Dose_Pump_Cmd )
      { S7_Templates := "SrcType := Real" } LT_Contact(in1 := "Totalizer_FT-04.01".value, in2 := #Param.min_Flow.ChiliAwetan3)
      { S7_Templates := "time_type := Time" } #Param.timerMon.ChiliAwetan3.TON(pt := #Param.timerMon.ChiliAwetan3.PT, et =>)
   END_RUNG
   RUNG wire#w1
      Contact( #Param.timerMon.ChiliAwetan3.Q )
      S_Coil( #AlarmFlow_Blend.%X2 )
   END_RUNG
   // the same network as SCL:
   #Param.timerMon.ChiliAwetan3.TON(IN := #alwaysON AND "T-04_ChiliAwetan_3".IN_Dose_Run AND NOT "T-04_ChiliAwetan_3".IN_Dose_Held AND "T-04_ChiliAwetan_3".IN_Dose_Pump_Cmd AND ("Totalizer_FT-04.01".value < #Param.min_Flow.ChiliAwetan3),
                           PT := #Param.timerMon.ChiliAwetan3.PT);
   IF #alwaysON AND #Param.timerMon.ChiliAwetan3.Q THEN #AlarmFlow_Blend.%X2 := TRUE; END_IF;
END_REGION

REGION Network 6: Alarm Flow Tomato
   RUNG wire#powerrail
      Contact( #alwaysON )
      wire#w1
      Contact( "T-05_Tomato".IN_Dose_Run )
      I_Contact( "T-05_Tomato".IN_Dose_Held )
      Contact( "T-05_Tomato".IN_Dose_Pump_Cmd )
      { S7_Templates := "SrcType := Real" } LT_Contact(in1 := "Totalizer_FT-05.01".value, in2 := #Param.min_Flow.Tomato)
      { S7_Templates := "time_type := Time" } #Param.timerMon.Tomato.TON(pt := #Param.timerMon.Tomato.PT, et =>)
   END_RUNG
   RUNG wire#w1
      Contact( #Param.timerMon.Tomato.Q )
      S_Coil( #AlarmFlow_Blend.%X3 )
   END_RUNG
   // the same network as SCL:
   #Param.timerMon.Tomato.TON(IN := #alwaysON AND "T-05_Tomato".IN_Dose_Run AND NOT "T-05_Tomato".IN_Dose_Held AND "T-05_Tomato".IN_Dose_Pump_Cmd AND ("Totalizer_FT-05.01".value < #Param.min_Flow.Tomato),
                           PT := #Param.timerMon.Tomato.PT);
   IF #alwaysON AND #Param.timerMon.Tomato.Q THEN #AlarmFlow_Blend.%X3 := TRUE; END_IF;
END_REGION

REGION Network 7: Alarm Flow ChiliFresh 1
   RUNG wire#powerrail
      Contact( #alwaysON )
      wire#w1
      Contact( "T-06_ChiliFresh_1".IN_Dose_Run )
      I_Contact( "T-06_ChiliFresh_1".IN_Dose_Held )
      Contact( "T-06_ChiliFresh_1".IN_Dose_Pump_Cmd )
      { S7_Templates := "SrcType := Real" } LT_Contact(in1 := "Totalizer_FT-06.01".value, in2 := #Param.min_Flow.ChiliFresh1)
      { S7_Templates := "time_type := Time" } #Param.timerMon.ChiliFresh1.TON(pt := #Param.timerMon.ChiliFresh1.PT, et =>)
   END_RUNG
   RUNG wire#w1
      Contact( #Param.timerMon.ChiliFresh1.Q )
      S_Coil( #AlarmFlow_Blend.%X4 )
   END_RUNG
   // the same network as SCL:
   #Param.timerMon.ChiliFresh1.TON(IN := #alwaysON AND "T-06_ChiliFresh_1".IN_Dose_Run AND NOT "T-06_ChiliFresh_1".IN_Dose_Held AND "T-06_ChiliFresh_1".IN_Dose_Pump_Cmd AND ("Totalizer_FT-06.01".value < #Param.min_Flow.ChiliFresh1),
                           PT := #Param.timerMon.ChiliFresh1.PT);
   IF #alwaysON AND #Param.timerMon.ChiliFresh1.Q THEN #AlarmFlow_Blend.%X4 := TRUE; END_IF;
END_REGION

REGION Network 8: Alarm Flow ChiliFresh 2
